LIN {X 0,Y 387.614,Z 136.056,A -85,B 0,C 180,E1 -14314.941,E2 -14314.941} C_VEL
LIN {X 0,Y 385.469,Z 134.733,A -85,B 0,C 180,E1 -14316.684,E2 -14316.684} C_VEL
LIN {X 0,Y 383.225,Z 132.712,A -85,B 0,C 180,E1 -14318.163,E2 -14318.163} C_VEL
LIN {X 0,Y 380.546,Z 129.667,A -85,B 0,C 180,E1 -14319.669,E2 -14319.669} C_VEL
LIN {X 0,Y 377.535,Z 127.903,A -85,B 0,C 180,E1 -14321.039,E2 -14321.039} C_VEL
LIN {X 0,Y 374.064,Z 124.674,A -85,B 0,C 180,E1 -14322.478,E2 -14322.478} C_VEL
LIN {X 0,Y 371.833,Z 122.319,A -85,B 0,C 180,E1 -14323.337,E2 -14323.337} C_VEL
LIN {X 0,Y 368.144,Z 119.325,A -85,B 0,C 180,E1 -14324.584,E2 -14324.584} C_VEL
LIN {X 0,Y 364.871,Z 115.734,A -85,B 0,C 180,E1 -14325.644,E2 -14325.644} C_VEL
LIN {X 0,Y 361.202,Z 112.484,A -85,B 0,C 180,E1 -14326.737,E2 -14326.737} C_VEL
LIN {X 0,Y 358.552,Z 109.441,A -85,B 0,C 180,E1 -14327.482,E2 -14327.482} C_VEL
LIN {X 0,Y 355.376,Z 106.45,A -85,B 0,C 180,E1 -14328.333,E2 -14328.333} C_VEL
LIN {X 0,Y 353.051,Z 103.518,A -85,B 0,C 180,E1 -14328.941,E2 -14328.941} C_VEL
LIN {X 0,Y 350.141,Z 100.557,A -85,B 0,C 180,E1 -14329.672,E2 -14329.672} C_VEL
LIN {X 0,Y 348.213,Z 97.966,A -85,B 0,C 180,E1 -14330.137,E2 -14330.137} C_VEL
LIN {X 0,Y 345.498,Z 95.057,A -85,B 0,C 180,E1 -14330.785,E2 -14330.785} C_VEL
LIN {X 0,Y 344.014,Z 92.683,A -85,B 0,C 180,E1 -14331.145,E2 -14331.145} C_VEL
LIN {X 0,Y 341.721,Z 90.357,A -85,B 0,C 180,E1 -14331.634,E2 -14331.634} C_VEL
LIN {X 0,Y 340.82,Z 88.079,A -85,B 0,C 180,E1 -14331.984,E2 -14331.984} C_VEL
LIN {X 0,Y 340.743,Z 87.555,A -85,B 0,C 180,E1 -14332.43,E2 -14332.43} C_VEL
LIN {X 0,Y 340.769,Z 87.54,A -85,B 0,C 180,E1 -14335.665,E2 -14335.665} C_VEL
LIN {X 0,Y 340.724,Z 87.528,A -85,B 0,C 180,E1 -14338.321,E2 -14338.321} C_VEL
LIN {X 0,Y 340.694,Z 87.545,A -85,B 0,C 180,E1 -14341.045,E2 -14341.045} C_VEL
LIN {X 0,Y 340.715,Z 87.514,A -85,B 0,C 180,E1 -14345.279,E2 -14345.279} C_VEL
LIN {X 0,Y 340.707,Z 87.545,A -85,B 0,C 180,E1 -14348.386,E2 -14348.386} C_VEL
LIN {X 0,Y 340.695,Z 87.5,A -85,B 0,C 180,E1 -14352.046,E2 -14352.046} C_VEL
LIN {X 0,Y 340.653,Z 87.551,A -85,B 0,C 180,E1 -14356.226,E2 -14356.226} C_VEL
LIN {X 0,Y 340.701,Z 87.535,A -85,B 0,C 180,E1 -14358.694,E2 -14358.694} C_VEL
LIN {X 0,Y 340.736,Z 87.543,A -85,B 0,C 180,E1 -14361.774,E2 -14361.774} C_VEL
LIN {X 0,Y 340.72,Z 87.526,A -85,B 0,C 180,E1 -14365.596,E2 -14365.596} C_VEL
LIN {X 0,Y 340.702,Z 87.543,A -85,B 0,C 180,E1 -14369.553,E2 -14369.553} C_VEL
LIN {X 0,Y 340.801,Z 87.511,A -85,B 0,C 180,E1 -14373.02,E2 -14373.02} C_VEL
LIN {X 0,Y 340.759,Z 87.528,A -85,B 0,C 180,E1 -14374.683,E2 -14374.683} C_VEL
LIN {X 0,Y 340.077,Z 87.623,A -85,B 0,C 180,E1 -14375.67,E2 -14375.67} C_VEL
LIN {X 0,Y 337.182,Z 87.982,A -85,B 0,C 180,E1 -14377.275,E2 -14377.275} C_VEL
LIN {X 0,Y 334.76,Z 88.277,A -85,B 0,C 180,E1 -14378.575,E2 -14378.575} C_VEL
LIN {X 0,Y 333.76,Z 88.394,A -85,B 0,C 180,E1 -14379.581,E2 -14379.581} C_VEL
LIN {X 0,Y 333.7,Z 88.393,A -85,B 0,C 180,E1 -14379.922,E2 -14379.922} C_VEL
LIN {X 0,Y 333.745,Z 88.397,A -85,B 0,C 180,E1 -14382.854,E2 -14382.854} C_VEL
LIN {X 0,Y 333.797,Z 88.402,A -85,B 0,C 180,E1 -14386.609,E2 -14386.609} C_VEL
LIN {X 0,Y 333.863,Z 88.365,A -85,B 0,C 180,E1 -14390.306,E2 -14390.306} C_VEL
LIN {X 0,Y 334.025,Z 88.368,A -85,B 0,C 180,E1 -14392.748,E2 -14392.748} C_VEL
LIN {X 0,Y 333.81,Z 88.402,A -85,B 0,C 180,E1 -14395.17,E2 -14395.17} C_VEL
LIN {X 0,Y 334.105,Z 88.355,A -85,B 0,C 180,E1 -14397.589,E2 -14397.589} C_VEL
LIN {X 0,Y 334.227,Z 88.319,A -85,B 0,C 180,E1 -14400.001,E2 -14400.001} C_VEL
LIN {X 0,Y 334.105,Z 88.356,A -85,B 0,C 180,E1 -14402.412,E2 -14402.412} C_VEL
LIN {X 0,Y 334.023,Z 88.374,A -85,B 0,C 180,E1 -14406.039,E2 -14406.039} C_VEL
LIN {X 0,Y 333.985,Z 88.358,A -85,B 0,C 180,E1 -14408.502,E2 -14408.502} C_VEL
LIN {X 0,Y 333.792,Z 88.395,A -85,B 0,C 180,E1 -14412.155,E2 -14412.155} C_VEL
LIN {X 0,Y 333.779,Z 88.399,A -85,B 0,C 180,E1 -14415.887,E2 -14415.887} C_VEL
LIN {X 0,Y 333.797,Z 88.374,A -85,B 0,C 180,E1 -14418.655,E2 -14418.655} C_VEL
LIN {X 0,Y 333.694,Z 88.414,A -85,B 0,C 180,E1 -14422.279,E2 -14422.279} C_VEL
LIN {X 0,Y 333.736,Z 88.392,A -85,B 0,C 180,E1 -14426.247,E2 -14426.247} C_VEL
LIN {X 0,Y 333.691,Z 88.409,A -85,B 0,C 180,E1 -14428.975,E2 -14428.975} C_VEL
LIN {X 0,Y 333.644,Z 88.417,A -85,B 0,C 180,E1 -14432.587,E2 -14432.587} C_VEL
LIN {X 0,Y 333.677,Z 88.415,A -85,B 0,C 180,E1 -14436.14,E2 -14436.14} C_VEL
LIN {X 0,Y 333.648,Z 88.414,A -85,B 0,C 180,E1 -14439.193,E2 -14439.193} C_VEL
LIN {X 0,Y 333.634,Z 88.428,A -85,B 0,C 180,E1 -14442.501,E2 -14442.501} C_VEL
LIN {X 0,Y 333.598,Z 88.427,A -85,B 0,C 180,E1 -14445.955,E2 -14445.955} C_VEL
LIN {X 0,Y 333.649,Z 88.399,A -85,B 0,C 180,E1 -14449.316,E2 -14449.316} C_VEL
LIN {X 0,Y 333.669,Z 88.419,A -85,B 0,C 180,E1 -14453.168,E2 -14453.168} C_VEL
LIN {X 0,Y 333.706,Z 88.483,A -85,B 0,C 180,E1 -14456.886,E2 -14456.886} C_VEL
LIN {X 0,Y 334.983,Z 94.79,A -85,B 0,C 180,E1 -14459.339,E2 -14459.339} C_VEL
LIN {X 0,Y 336.52,Z 102.522,A -85,B 0,C 180,E1 -14462.042,E2 -14462.042} C_VEL
LIN {X 0,Y 337.063,Z 107.291,A -85,B 0,C 180,E1 -14463.713,E2 -14463.713} C_VEL
LIN {X 0,Y 336.216,Z 114.217,A -85,B 0,C 180,E1 -14465.934,E2 -14465.934} C_VEL
LIN {X 0,Y 337.962,Z 122.359,A -85,B 0,C 180,E1 -14466.298,E2 -14466.298} C_VEL
LIN {X 0,Y 342.357,Z 144.864,A -85,B 0,C 180,E1 -14467.12,E2 -14467.12} C_VEL
LIN {X 0,Y 343.665,Z 153.202,A -85,B 0,C 180,E1 -14467.396,E2 -14467.396} C_VEL
LIN {X 0,Y 342.418,Z 218.942,A -85,B 0,C 180,E1 -14468.793,E2 -14468.793} C_VEL
LIN {X 0,Y 341.88,Z 229.679,A -85,B 0,C 180,E1 -14469.152,E2 -14469.152} C_VEL
LIN {X 0,Y 341.203,Z 238.778,A -85,B 0,C 180,E1 -14469.582,E2 -14469.582} C_VEL
LIN {X 0,Y 340.4,Z 248.132,A -85,B 0,C 180,E1 -14470.161,E2 -14470.161} C_VEL
LIN {X 0,Y 339.412,Z 258.273,A -85,B 0,C 180,E1 -14470.966,E2 -14470.966} C_VEL
LIN {X 0,Y 338.345,Z 267.266,A -85,B 0,C 180,E1 -14471.846,E2 -14471.846} C_VEL
LIN {X 0,Y 337.271,Z 275.994,A -85,B 0,C 180,E1 -14472.882,E2 -14472.882} C_VEL
LIN {X 0,Y 336.259,Z 283.752,A -85,B 0,C 180,E1 -14473.982,E2 -14473.982} C_VEL
LIN {X 0,Y 335.422,Z 290.636,A -85,B 0,C 180,E1 -14475.133,E2 -14475.133} C_VEL
LIN {X 0,Y 334.663,Z 296.812,A -85,B 0,C 180,E1 -14476.335,E2 -14476.335} C_VEL
LIN {X 0,Y 333.727,Z 303.347,A -85,B 0,C 180,E1 -14477.843,E2 -14477.843} C_VEL
LIN {X 0,Y 333.206,Z 307.85,A -85,B 0,C 180,E1 -14479.057,E2 -14479.057} C_VEL
LIN {X 0,Y 332.602,Z 313.342,A -85,B 0,C 180,E1 -14480.881,E2 -14480.881} C_VEL
LIN {X 0,Y 332.201,Z 317.667,A -85,B 0,C 180,E1 -14482.708,E2 -14482.708} C_VEL
LIN {X 0,Y 332.028,Z 320.418,A -85,B 0,C 180,E1 -14484.183,E2 -14484.183} C_VEL
LIN {X 0,Y 331.969,Z 323.224,A -85,B 0,C 180,E1 -14486.359,E2 -14486.359} C_VEL
LIN {X 0,Y 331.916,Z 324.281,A -85,B 0,C 180,E1 -14487.573,E2 -14487.573} C_VEL
LIN {X 0,Y 331.913,Z 324.87,A -85,B 0,C 180,E1 -14488.787,E2 -14488.787} C_VEL
LIN {X 0,Y 331.97,Z 325.026,A -85,B 0,C 180,E1 -14490,E2 -14490} C_VEL
LIN {X 0,Y 331.913,Z 324.87,A -85,B 0,C 180,E1 -14491.213,E2 -14491.213} C_VEL
LIN {X 0,Y 331.916,Z 324.281,A -85,B 0,C 180,E1 -14492.427,E2 -14492.427} C_VEL
LIN {X 0,Y 331.969,Z 321.835,A -85,B 0,C 180,E1 -14494.858,E2 -14494.858} C_VEL
LIN {X 0,Y 332.11,Z 318.884,A -85,B 0,C 180,E1 -14496.684,E2 -14496.684} C_VEL
LIN {X 0,Y 332.46,Z 314.897,A -85,B 0,C 180,E1 -14498.51,E2 -14498.51} C_VEL
LIN {X 0,Y 332.971,Z 309.766,A -85,B 0,C 180,E1 -14500.335,E2 -14500.335} C_VEL
LIN {X 0,Y 333.566,Z 304.502,A -85,B 0,C 180,E1 -14501.854,E2 -14501.854} C_VEL
LIN {X 0,Y 334.462,Z 298.188,A -85,B 0,C 180,E1 -14503.364,E2 -14503.364} C_VEL
LIN {X 0,Y 335.206,Z 292.235,A -85,B 0,C 180,E1 -14504.572,E2 -14504.572} C_VEL
LIN {X 0,Y 336.181,Z 285.31,A -85,B 0,C 180,E1 -14505.77,E2 -14505.77} C_VEL
LIN {X 0,Y 337.15,Z 277.129,A -85,B 0,C 180,E1 -14506.968,E2 -14506.968} C_VEL
LIN {X 0,Y 338.211,Z 268.619,A -85,B 0,C 180,E1 -14508.005,E2 -14508.005} C_VEL
LIN {X 0,Y 339.257,Z 259.905,A -85,B 0,C 180,E1 -14508.886,E2 -14508.886} C_VEL
LIN {X 0,Y 340.232,Z 250.147,A -85,B 0,C 180,E1 -14509.692,E2 -14509.692} C_VEL
LIN {X 0,Y 341.021,Z 241.354,A -85,B 0,C 180,E1 -14510.272,E2 -14510.272} C_VEL
LIN {X 0,Y 341.773,Z 231.427,A -85,B 0,C 180,E1 -14510.776,E2 -14510.776} C_VEL
LIN {X 0,Y 342.274,Z 221.571,A -85,B 0,C 180,E1 -14511.138,E2 -14511.138} C_VEL
LIN {X 0,Y 342.869,Z 198.751,A -85,B 0,C 180,E1 -14511.651,E2 -14511.651} C_VEL
LIN {X 0,Y 343.58,Z 152.553,A -85,B 0,C 180,E1 -14512.624,E2 -14512.624} C_VEL
LIN {X 0,Y 339.442,Z 129.203,A -85,B 0,C 180,E1 -14513.439,E2 -14513.439} C_VEL
LIN {X 0,Y 336.241,Z 114.522,A -85,B 0,C 180,E1 -14514.032,E2 -14514.032} C_VEL
LIN {X 0,Y 336.325,Z 112.923,A -85,B 0,C 180,E1 -14514.408,E2 -14514.408} C_VEL
LIN {X 0,Y 337.068,Z 107.285,A -85,B 0,C 180,E1 -14516.288,E2 -14516.288} C_VEL
LIN {X 0,Y 336.514,Z 102.53,A -85,B 0,C 180,E1 -14517.956,E2 -14517.956} C_VEL
LIN {X 0,Y 334.834,Z 93.824,A -85,B 0,C 180,E1 -14521.091,E2 -14521.091} C_VEL
LIN {X 0,Y 333.676,Z 88.433,A -85,B 0,C 180,E1 -14523.161,E2 -14523.161} C_VEL
LIN {X 0,Y 333.669,Z 88.419,A -85,B 0,C 180,E1 -14526.832,E2 -14526.832} C_VEL
LIN {X 0,Y 333.648,Z 88.4,A -85,B 0,C 180,E1 -14530.767,E2 -14530.767} C_VEL
LIN {X 0,Y 333.595,Z 88.428,A -85,B 0,C 180,E1 -14534.25,E2 -14534.25} C_VEL
LIN {X 0,Y 333.643,Z 88.426,A -85,B 0,C 180,E1 -14537.618,E2 -14537.618} C_VEL
LIN {X 0,Y 333.654,Z 88.417,A -85,B 0,C 180,E1 -14541.202,E2 -14541.202} C_VEL
LIN {X 0,Y 333.677,Z 88.415,A -85,B 0,C 180,E1 -14543.86,E2 -14543.86} C_VEL
LIN {X 0,Y 333.644,Z 88.417,A -85,B 0,C 180,E1 -14547.413,E2 -14547.413} C_VEL
LIN {X 0,Y 333.691,Z 88.409,A -85,B 0,C 180,E1 -14551.025,E2 -14551.025} C_VEL
LIN {X 0,Y 333.736,Z 88.392,A -85,B 0,C 180,E1 -14553.753,E2 -14553.753} C_VEL
LIN {X 0,Y 333.721,Z 88.411,A -85,B 0,C 180,E1 -14557.913,E2 -14557.913} C_VEL
LIN {X 0,Y 333.794,Z 88.375,A -85,B 0,C 180,E1 -14561.589,E2 -14561.589} C_VEL
LIN {X 0,Y 333.809,Z 88.4,A -85,B 0,C 180,E1 -14565.576,E2 -14565.576} C_VEL
LIN {X 0,Y 333.834,Z 88.376,A -85,B 0,C 180,E1 -14569.077,E2 -14569.077} C_VEL
LIN {X 0,Y 334.027,Z 88.366,A -85,B 0,C 180,E1 -14572.747,E2 -14572.747} C_VEL
LIN {X 0,Y 333.812,Z 88.402,A -85,B 0,C 180,E1 -14575.168,E2 -14575.168} C_VEL
LIN {X 0,Y 334.105,Z 88.356,A -85,B 0,C 180,E1 -14577.588,E2 -14577.588} C_VEL
LIN {X 0,Y 334.227,Z 88.319,A -85,B 0,C 180,E1 -14579.999,E2 -14579.999} C_VEL
LIN {X 0,Y 334.105,Z 88.355,A -85,B 0,C 180,E1 -14582.411,E2 -14582.411} C_VEL
LIN {X 0,Y 334.025,Z 88.368,A -85,B 0,C 180,E1 -14587.252,E2 -14587.252} C_VEL
LIN {X 0,Y 333.836,Z 88.376,A -85,B 0,C 180,E1 -14590.921,E2 -14590.921} C_VEL
LIN {X 0,Y 333.807,Z 88.403,A -85,B 0,C 180,E1 -14594.634,E2 -14594.634} C_VEL
LIN {X 0,Y 333.794,Z 88.378,A -85,B 0,C 180,E1 -14598.654,E2 -14598.654} C_VEL
LIN {X 0,Y 333.691,Z 88.416,A -85,B 0,C 180,E1 -14602.278,E2 -14602.278} C_VEL
LIN {X 0,Y 333.733,Z 88.397,A -85,B 0,C 180,E1 -14606.246,E2 -14606.246} C_VEL
LIN {X 0,Y 333.687,Z 88.408,A -85,B 0,C 180,E1 -14608.973,E2 -14608.973} C_VEL
LIN {X 0,Y 333.64,Z 88.42,A -85,B 0,C 180,E1 -14612.586,E2 -14612.586} C_VEL
LIN {X 0,Y 333.674,Z 88.414,A -85,B 0,C 180,E1 -14616.138,E2 -14616.138} C_VEL
LIN {X 0,Y 333.669,Z 88.415,A -85,B 0,C 180,E1 -14619.188,E2 -14619.188} C_VEL
LIN {X 0,Y 333.657,Z 88.421,A -85,B 0,C 180,E1 -14622.505,E2 -14622.505} C_VEL
LIN {X 0,Y 333.593,Z 88.405,A -85,B 0,C 180,E1 -14625.955,E2 -14625.955} C_VEL
LIN {X 0,Y 333.643,Z 88.39,A -85,B 0,C 180,E1 -14629.315,E2 -14629.315} C_VEL
LIN {X 0,Y 333.662,Z 88.419,A -85,B 0,C 180,E1 -14633.167,E2 -14633.167} C_VEL
LIN {X 0,Y 333.67,Z 88.39,A -85,B 0,C 180,E1 -14635.341,E2 -14635.341} C_VEL
LIN {X 0,Y 333.686,Z 88.405,A -85,B 0,C 180,E1 -14639.637,E2 -14639.637} C_VEL
LIN {X 0,Y 333.736,Z 88.41,A -85,B 0,C 180,E1 -14642.401,E2 -14642.401} C_VEL
LIN {X 0,Y 333.723,Z 88.417,A -85,B 0,C 180,E1 -14645.091,E2 -14645.091} C_VEL
LIN {X 0,Y 333.715,Z 88.563,A -85,B 0,C 180,E1 -14646.635,E2 -14646.635} C_VEL
LIN {X 0,Y 333.903,Z 89.473,A -85,B 0,C 180,E1 -14646.906,E2 -14646.906} C_VEL
LIN {X 0,Y 335.441,Z 92.245,A -85,B 0,C 180,E1 -14647.293,E2 -14647.293} C_VEL
LIN {X 0,Y 337.24,Z 94.134,A -85,B 0,C 180,E1 -14647.649,E2 -14647.649} C_VEL
LIN {X 0,Y 339.457,Z 97.377,A -85,B 0,C 180,E1 -14648.16,E2 -14648.16} C_VEL
LIN {X 0,Y 341.244,Z 99.3,A -85,B 0,C 180,E1 -14648.55,E2 -14648.55} C_VEL
LIN {X 0,Y 344.183,Z 103.016,A -85,B 0,C 180,E1 -14649.205,E2 -14649.205} C_VEL
LIN {X 0,Y 346.131,Z 105.087,A -85,B 0,C 180,E1 -14649.669,E2 -14649.669} C_VEL
LIN {X 0,Y 349.254,Z 108.734,A -85,B 0,C 180,E1 -14650.409,E2 -14650.409} C_VEL
LIN {X 0,Y 351.181,Z 110.612,A -85,B 0,C 180,E1 -14650.88,E2 -14650.88} C_VEL
LIN {X 0,Y 354.741,Z 114.632,A -85,B 0,C 180,E1 -14651.8,E2 -14651.8} C_VEL
LIN {X 0,Y 357.121,Z 116.838,A -85,B 0,C 180,E1 -14652.431,E2 -14652.431} C_VEL
LIN {X 0,Y 361.089,Z 120.94,A -85,B 0,C 180,E1 -14653.544,E2 -14653.544} C_VEL
LIN {X 0,Y 363.83,Z 123.291,A -85,B 0,C 180,E1 -14654.364,E2 -14654.364} C_VEL
LIN {X 0,Y 367.524,Z 127.112,A -85,B 0,C 180,E1 -14655.553,E2 -14655.553} C_VEL
LIN {X 0,Y 371.229,Z 130.062,A -85,B 0,C 180,E1 -14656.813,E2 -14656.813} C_VEL
LIN {X 0,Y 374.888,Z 133.747,A -85,B 0,C 180,E1 -14658.241,E2 -14658.241} C_VEL
LIN {X 0,Y 378.478,Z 136.219,A -85,B 0,C 180,E1 -14659.786,E2 -14659.786} C_VEL
LIN {X 0,Y 379.78,Z 137.046,A -85,B 0,C 180,E1 -14660.413,E2 -14660.413} C_VEL
LIN {X 0,Y 382.384,Z 139.979,A -85,B 0,C 180,E1 -14661.881,E2 -14661.881} C_VEL
LIN {X 0,Y 384.713,Z 141.903,A -85,B 0,C 180,E1 -14663.407,E2 -14663.407} C_VEL
LIN {X 0,Y 387.037,Z 143.23,A -85,B 0,C 180,E1 -14665.318,E2 -14665.318} C_VEL
LIN {X 0,Y 388.665,Z 143.823,A -85,B 0,C 180,E1 -14667.428,E2 -14667.428} C_VEL
LIN {X 0,Y 389.264,Z 144.277,A -85,B 0,C 180,E1 -14668.965,E2 -14668.965} C_VEL
LIN {X 0,Y 389.407,Z 144.179,A -85,B 0,C 180,E1 -14670,E2 -14670} C_VEL
LIN {X 0,Y 389.126,Z 144.135,A -85,B 0,C 180,E1 -14671.552,E2 -14671.552} C_VEL
LIN {X 0,Y 388.36,Z 143.701,A -85,B 0,C 180,E1 -14673.112,E2 -14673.112} C_VEL
LIN {X 0,Y 386.736,Z 143.092,A -85,B 0,C 180,E1 -14674.943,E2 -14674.943} C_VEL
LIN {X 0,Y 384.56,Z 141.783,A -85,B 0,C 180,E1 -14676.7,E2 -14676.7} C_VEL
LIN {X 0,Y 382.221,Z 139.834,A -85,B 0,C 180,E1 -14678.214,E2 -14678.214} C_VEL
LIN {X 0,Y 379.214,Z 136.56,A -85,B 0,C 180,E1 -14679.864,E2 -14679.864} C_VEL
LIN {X 0,Y 376.134,Z 134.752,A -85,B 0,C 180,E1 -14681.228,E2 -14681.228} C_VEL
LIN {X 0,Y 372.666,Z 131.662,A -85,B 0,C 180,E1 -14682.629,E2 -14682.629} C_VEL
LIN {X 0,Y 370.003,Z 128.94,A -85,B 0,C 180,E1 -14683.635,E2 -14683.635} C_VEL
LIN {X 0,Y 366.039,Z 125.687,A -85,B 0,C 180,E1 -14684.945,E2 -14684.945} C_VEL
LIN {X 0,Y 362.682,Z 122.188,A -85,B 0,C 180,E1 -14685.986,E2 -14685.986} C_VEL
LIN {X 0,Y 358.732,Z 118.722,A -85,B 0,C 180,E1 -14687.109,E2 -14687.109} C_VEL
LIN {X 0,Y 355.813,Z 115.508,A -85,B 0,C 180,E1 -14687.929,E2 -14687.929} C_VEL
LIN {X 0,Y 352.189,Z 111.983,A -85,B 0,C 180,E1 -14688.848,E2 -14688.848} C_VEL
LIN {X 0,Y 350.013,Z 109.386,A -85,B 0,C 180,E1 -14689.415,E2 -14689.415} C_VEL
LIN {X 0,Y 346.456,Z 105.581,A -85,B 0,C 180,E1 -14690.25,E2 -14690.25} C_VEL
LIN {X 0,Y 344.965,Z 103.745,A -85,B 0,C 180,E1 -14690.614,E2 -14690.614} C_VEL
LIN {X 0,Y 341.952,Z 100.422,A -85,B 0,C 180,E1 -14691.286,E2 -14691.286} C_VEL
LIN {X 0,Y 340.285,Z 98.185,A -85,B 0,C 180,E1 -14691.661,E2 -14691.661} C_VEL
LIN {X 0,Y 337.761,Z 95.054,A -85,B 0,C 180,E1 -14692.231,E2 -14692.231} C_VEL
LIN {X 0,Y 336.543,Z 93.281,A -85,B 0,C 180,E1 -14692.493,E2 -14692.493} C_VEL
LIN {X 0,Y 334.617,Z 91.122,A -85,B 0,C 180,E1 -14692.878,E2 -14692.878} C_VEL
LIN {X 0,Y 333.802,Z 89.069,A -85,B 0,C 180,E1 -14693.171,E2 -14693.171} C_VEL
LIN {X 0,Y 333.68,Z 88.493,A -85,B 0,C 180,E1 -14693.425,E2 -14693.425} C_VEL
LIN {X 0,Y 333.731,Z 88.416,A -85,B 0,C 180,E1 -14696.247,E2 -14696.247} C_VEL
LIN {X 0,Y 333.686,Z 88.399,A -85,B 0,C 180,E1 -14698.974,E2 -14698.974} C_VEL
LIN {X 0,Y 333.64,Z 88.421,A -85,B 0,C 180,E1 -14702.587,E2 -14702.587} C_VEL
LIN {X 0,Y 333.673,Z 88.401,A -85,B 0,C 180,E1 -14706.139,E2 -14706.139} C_VEL
LIN {X 0,Y 333.643,Z 88.418,A -85,B 0,C 180,E1 -14709.193,E2 -14709.193} C_VEL
LIN {X 0,Y 333.628,Z 88.381,A -85,B 0,C 180,E1 -14712.5,E2 -14712.5} C_VEL
LIN {X 0,Y 333.597,Z 88.431,A -85,B 0,C 180,E1 -14715.956,E2 -14715.956} C_VEL
LIN {X 0,Y 333.653,Z 88.41,A -85,B 0,C 180,E1 -14719.314,E2 -14719.314} C_VEL
LIN {X 0,Y 333.653,Z 88.424,A -85,B 0,C 180,E1 -14722.35,E2 -14722.35} C_VEL
LIN {X 0,Y 333.671,Z 88.403,A -85,B 0,C 180,E1 -14725.342,E2 -14725.342} C_VEL
LIN {X 0,Y 333.688,Z 88.418,A -85,B 0,C 180,E1 -14729.638,E2 -14729.638} C_VEL
LIN {X 0,Y 333.737,Z 88.391,A -85,B 0,C 180,E1 -14732.401,E2 -14732.401} C_VEL
LIN {X 0,Y 333.725,Z 88.409,A -85,B 0,C 180,E1 -14735.091,E2 -14735.091} C_VEL
LIN {X 0,Y 333.678,Z 88.407,A -85,B 0,C 180,E1 -14739.02,E2 -14739.02} C_VEL
LIN {X 0,Y 333.7,Z 88.393,A -85,B 0,C 180,E1 -14739.922,E2 -14739.922} C_VEL
LIN {X 0,Y 333.09,Z 88.468,A -85,B 0,C 180,E1 -14740.929,E2 -14740.929} C_VEL
LIN {X 0,Y 330.266,Z 88.832,A -85,B 0,C 180,E1 -14742.568,E2 -14742.568} C_VEL
LIN {X 0,Y 327.852,Z 89.143,A -85,B 0,C 180,E1 -14743.896,E2 -14743.896} C_VEL
LIN {X 0,Y 326.83,Z 89.274,A -85,B 0,C 180,E1 -14744.924,E2 -14744.924} C_VEL
LIN {X 0,Y 326.756,Z 89.282,A -85,B 0,C 180,E1 -14745.272,E2 -14745.272} C_VEL
LIN {X 0,Y 326.772,Z 89.256,A -85,B 0,C 180,E1 -14748.84,E2 -14748.84} C_VEL
LIN {X 0,Y 326.979,Z 89.242,A -85,B 0,C 180,E1 -14752.591,E2 -14752.591} C_VEL
LIN {X 0,Y 326.777,Z 89.278,A -85,B 0,C 180,E1 -14755.066,E2 -14755.066} C_VEL
LIN {X 0,Y 327.046,Z 89.234,A -85,B 0,C 180,E1 -14757.537,E2 -14757.537} C_VEL
LIN {X 0,Y 327.179,Z 89.196,A -85,B 0,C 180,E1 -14760.001,E2 -14760.001} C_VEL
LIN {X 0,Y 327.046,Z 89.236,A -85,B 0,C 180,E1 -14762.464,E2 -14762.464} C_VEL
LIN {X 0,Y 326.999,Z 89.247,A -85,B 0,C 180,E1 -14766.17,E2 -14766.17} C_VEL
LIN {X 0,Y 326.915,Z 89.236,A -85,B 0,C 180,E1 -14768.656,E2 -14768.656} C_VEL
LIN {X 0,Y 326.736,Z 89.277,A -85,B 0,C 180,E1 -14772.422,E2 -14772.422} C_VEL
LIN {X 0,Y 326.755,Z 89.28,A -85,B 0,C 180,E1 -14774.958,E2 -14774.958} C_VEL
LIN {X 0,Y 326.733,Z 89.253,A -85,B 0,C 180,E1 -14778.839,E2 -14778.839} C_VEL
LIN {X 0,Y 326.622,Z 89.297,A -85,B 0,C 180,E1 -14782.788,E2 -14782.788} C_VEL
LIN {X 0,Y 326.691,Z 89.274,A -85,B 0,C 180,E1 -14785.484,E2 -14785.484} C_VEL
LIN {X 0,Y 326.649,Z 89.295,A -85,B 0,C 180,E1 -14789.661,E2 -14789.661} C_VEL
LIN {X 0,Y 326.608,Z 89.28,A -85,B 0,C 180,E1 -14794.02,E2 -14794.02} C_VEL
LIN {X 0,Y 326.629,Z 89.299,A -85,B 0,C 180,E1 -14797.239,E2 -14797.239} C_VEL
LIN {X 0,Y 326.579,Z 89.297,A -85,B 0,C 180,E1 -14801.132,E2 -14801.132} C_VEL
LIN {X 0,Y 326.529,Z 89.303,A -85,B 0,C 180,E1 -14804.743,E2 -14804.743} C_VEL
LIN {X 0,Y 326.578,Z 89.293,A -85,B 0,C 180,E1 -14808.155,E2 -14808.155} C_VEL
LIN {X 0,Y 326.627,Z 89.285,A -85,B 0,C 180,E1 -14811.392,E2 -14811.392} C_VEL
LIN {X 0,Y 326.622,Z 89.283,A -85,B 0,C 180,E1 -14814.852,E2 -14814.852} C_VEL
LIN {X 0,Y 326.676,Z 89.534,A -85,B 0,C 180,E1 -14816.565,E2 -14816.565} C_VEL
LIN {X 0,Y 328.195,Z 96.942,A -85,B 0,C 180,E1 -14819.431,E2 -14819.431} C_VEL
LIN {X 0,Y 329.614,Z 104.093,A -85,B 0,C 180,E1 -14822.025,E2 -14822.025} C_VEL
LIN {X 0,Y 330.081,Z 108.039,A -85,B 0,C 180,E1 -14823.441,E2 -14823.441} C_VEL
LIN {X 0,Y 329.381,Z 113.892,A -85,B 0,C 180,E1 -14825.38,E2 -14825.38} C_VEL
LIN {X 0,Y 330.25,Z 118.246,A -85,B 0,C 180,E1 -14825.619,E2 -14825.619} C_VEL
LIN {X 0,Y 334.159,Z 136.803,A -85,B 0,C 180,E1 -14826.346,E2 -14826.346} C_VEL
LIN {X 0,Y 337.096,Z 153.67,A -85,B 0,C 180,E1 -14826.945,E2 -14826.945} C_VEL
LIN {X 0,Y 335.823,Z 218.758,A -85,B 0,C 180,E1 -14828.355,E2 -14828.355} C_VEL
LIN {X 0,Y 335.27,Z 229.489,A -85,B 0,C 180,E1 -14828.721,E2 -14828.721} C_VEL
LIN {X 0,Y 334.563,Z 238.588,A -85,B 0,C 180,E1 -14829.158,E2 -14829.158} C_VEL
LIN {X 0,Y 333.747,Z 247.942,A -85,B 0,C 180,E1 -14829.749,E2 -14829.749} C_VEL
LIN {X 0,Y 332.703,Z 258.082,A -85,B 0,C 180,E1 -14830.567,E2 -14830.567} C_VEL
LIN {X 0,Y 331.594,Z 267.076,A -85,B 0,C 180,E1 -14831.463,E2 -14831.463} C_VEL
LIN {X 0,Y 330.473,Z 275.803,A -85,B 0,C 180,E1 -14832.519,E2 -14832.519} C_VEL
LIN {X 0,Y 329.484,Z 283.197,A -85,B 0,C 180,E1 -14833.583,E2 -14833.583} C_VEL
LIN {X 0,Y 328.52,Z 290.62,A -85,B 0,C 180,E1 -14834.847,E2 -14834.847} C_VEL
LIN {X 0,Y 327.75,Z 296.621,A -85,B 0,C 180,E1 -14836.041,E2 -14836.041} C_VEL
LIN {X 0,Y 326.766,Z 303.156,A -85,B 0,C 180,E1 -14837.58,E2 -14837.58} C_VEL
LIN {X 0,Y 326.18,Z 307.658,A -85,B 0,C 180,E1 -14838.819,E2 -14838.819} C_VEL
LIN {X 0,Y 325.57,Z 313.151,A -85,B 0,C 180,E1 -14840.683,E2 -14840.683} C_VEL
LIN {X 0,Y 325.153,Z 317.477,A -85,B 0,C 180,E1 -14842.549,E2 -14842.549} C_VEL
LIN {X 0,Y 324.92,Z 320.521,A -85,B 0,C 180,E1 -14844.259,E2 -14844.259} C_VEL
LIN {X 0,Y 324.876,Z 323.033,A -85,B 0,C 180,E1 -14846.279,E2 -14846.279} C_VEL
LIN {X 0,Y 324.835,Z 324.091,A -85,B 0,C 180,E1 -14847.52,E2 -14847.52} C_VEL
LIN {X 0,Y 324.822,Z 324.68,A -85,B 0,C 180,E1 -14848.76,E2 -14848.76} C_VEL
LIN {X 0,Y 324.874,Z 324.836,A -85,B 0,C 180,E1 -14850,E2 -14850} C_VEL
LIN {X 0,Y 324.822,Z 324.68,A -85,B 0,C 180,E1 -14851.24,E2 -14851.24} C_VEL
LIN {X 0,Y 324.835,Z 324.091,A -85,B 0,C 180,E1 -14852.48,E2 -14852.48} C_VEL
LIN {X 0,Y 324.88,Z 321.644,A -85,B 0,C 180,E1 -14854.964,E2 -14854.964} C_VEL
LIN {X 0,Y 325.049,Z 318.694,A -85,B 0,C 180,E1 -14856.83,E2 -14856.83} C_VEL
LIN {X 0,Y 325.4,Z 314.705,A -85,B 0,C 180,E1 -14858.696,E2 -14858.696} C_VEL
LIN {X 0,Y 325.948,Z 309.574,A -85,B 0,C 180,E1 -14860.561,E2 -14860.561} C_VEL
LIN {X 0,Y 326.601,Z 304.311,A -85,B 0,C 180,E1 -14862.111,E2 -14862.111} C_VEL
LIN {X 0,Y 327.541,Z 297.997,A -85,B 0,C 180,E1 -14863.652,E2 -14863.652} C_VEL
LIN {X 0,Y 328.313,Z 292.044,A -85,B 0,C 180,E1 -14864.885,E2 -14864.885} C_VEL
LIN {X 0,Y 329.28,Z 285.118,A -85,B 0,C 180,E1 -14866.109,E2 -14866.109} C_VEL
LIN {X 0,Y 330.323,Z 276.937,A -85,B 0,C 180,E1 -14867.329,E2 -14867.329} C_VEL
LIN {X 0,Y 331.444,Z 268.428,A -85,B 0,C 180,E1 -14868.386,E2 -14868.386} C_VEL
LIN {X 0,Y 332.545,Z 259.714,A -85,B 0,C 180,E1 -14869.282,E2 -14869.282} C_VEL
LIN {X 0,Y 333.565,Z 249.957,A -85,B 0,C 180,E1 -14870.102,E2 -14870.102} C_VEL
LIN {X 0,Y 334.388,Z 241.164,A -85,B 0,C 180,E1 -14870.693,E2 -14870.693} C_VEL
LIN {X 0,Y 335.151,Z 231.237,A -85,B 0,C 180,E1 -14871.206,E2 -14871.206} C_VEL
LIN {X 0,Y 335.667,Z 221.381,A -85,B 0,C 180,E1 -14871.575,E2 -14871.575} C_VEL
LIN {X 0,Y 336.282,Z 198.56,A -85,B 0,C 180,E1 -14872.097,E2 -14872.097} C_VEL
LIN {X 0,Y 337.047,Z 153.551,A -85,B 0,C 180,E1 -14873.061,E2 -14873.061} C_VEL
LIN {X 0,Y 333.076,Z 131.136,A -85,B 0,C 180,E1 -14873.865,E2 -14873.865} C_VEL
LIN {X 0,Y 329.428,Z 114.114,A -85,B 0,C 180,E1 -14874.583,E2 -14874.583} C_VEL
LIN {X 0,Y 329.614,Z 111.881,A -85,B 0,C 180,E1 -14875.242,E2 -14875.242} C_VEL
LIN {X 0,Y 330.099,Z 107.941,A -85,B 0,C 180,E1 -14876.592,E2 -14876.592} C_VEL
LIN {X 0,Y 329.139,Z 101.587,A -85,B 0,C 180,E1 -14878.899,E2 -14878.899} C_VEL
LIN {X 0,Y 327.224,Z 92.007,A -85,B 0,C 180,E1 -14882.475,E2 -14882.475} C_VEL
LIN {X 0,Y 326.631,Z 89.312,A -85,B 0,C 180,E1 -14883.584,E2 -14883.584} C_VEL
LIN {X 0,Y 326.632,Z 89.299,A -85,B 0,C 180,E1 -14887.239,E2 -14887.239} C_VEL
LIN {X 0,Y 326.579,Z 89.283,A -85,B 0,C 180,E1 -14891.131,E2 -14891.131} C_VEL
LIN {X 0,Y 326.529,Z 89.305,A -85,B 0,C 180,E1 -14894.742,E2 -14894.742} C_VEL
LIN {X 0,Y 326.578,Z 89.303,A -85,B 0,C 180,E1 -14898.154,E2 -14898.154} C_VEL
LIN {X 0,Y 326.625,Z 89.295,A -85,B 0,C 180,E1 -14901.391,E2 -14901.391} C_VEL
LIN {X 0,Y 326.621,Z 89.284,A -85,B 0,C 180,E1 -14904.851,E2 -14904.851} C_VEL
LIN {X 0,Y 326.609,Z 89.294,A -85,B 0,C 180,E1 -14907.455,E2 -14907.455} C_VEL
LIN {X 0,Y 326.649,Z 89.295,A -85,B 0,C 180,E1 -14910.339,E2 -14910.339} C_VEL
LIN {X 0,Y 326.691,Z 89.274,A -85,B 0,C 180,E1 -14914.516,E2 -14914.516} C_VEL
LIN {X 0,Y 326.647,Z 89.288,A -85,B 0,C 180,E1 -14918.545,E2 -14918.545} C_VEL
LIN {X 0,Y 326.745,Z 89.251,A -85,B 0,C 180,E1 -14921.177,E2 -14921.177} C_VEL
LIN {X 0,Y 326.764,Z 89.278,A -85,B 0,C 180,E1 -14925.432,E2 -14925.432} C_VEL
LIN {X 0,Y 326.77,Z 89.257,A -85,B 0,C 180,E1 -14928.838,E2 -14928.838} C_VEL
LIN {X 0,Y 326.981,Z 89.24,A -85,B 0,C 180,E1 -14932.59,E2 -14932.59} C_VEL
LIN {X 0,Y 326.779,Z 89.278,A -85,B 0,C 180,E1 -14935.064,E2 -14935.064} C_VEL
LIN {X 0,Y 327.046,Z 89.236,A -85,B 0,C 180,E1 -14937.536,E2 -14937.536} C_VEL
LIN {X 0,Y 327.179,Z 89.196,A -85,B 0,C 180,E1 -14939.999,E2 -14939.999} C_VEL
LIN {X 0,Y 327.046,Z 89.234,A -85,B 0,C 180,E1 -14942.463,E2 -14942.463} C_VEL
LIN {X 0,Y 326.971,Z 89.246,A -85,B 0,C 180,E1 -14946.654,E2 -14946.654} C_VEL
LIN {X 0,Y 326.814,Z 89.242,A -85,B 0,C 180,E1 -14949.906,E2 -14949.906} C_VEL
LIN {X 0,Y 326.759,Z 89.283,A -85,B 0,C 180,E1 -14953.685,E2 -14953.685} C_VEL
LIN {X 0,Y 326.697,Z 89.27,A -85,B 0,C 180,E1 -14957.527,E2 -14957.527} C_VEL
LIN {X 0,Y 326.661,Z 89.273,A -85,B 0,C 180,E1 -14960.134,E2 -14960.134} C_VEL
LIN {X 0,Y 326.65,Z 89.293,A -85,B 0,C 180,E1 -14964.128,E2 -14964.128} C_VEL
LIN {X 0,Y 326.68,Z 89.269,A -85,B 0,C 180,E1 -14966.857,E2 -14966.857} C_VEL
LIN {X 0,Y 326.631,Z 89.298,A -85,B 0,C 180,E1 -14970.609,E2 -14970.609} C_VEL
LIN {X 0,Y 326.604,Z 89.284,A -85,B 0,C 180,E1 -14974.019,E2 -14974.019} C_VEL
LIN {X 0,Y 326.627,Z 89.301,A -85,B 0,C 180,E1 -14977.239,E2 -14977.239} C_VEL
LIN {X 0,Y 326.601,Z 89.289,A -85,B 0,C 180,E1 -14980.207,E2 -14980.207} C_VEL
LIN {X 0,Y 326.569,Z 89.305,A -85,B 0,C 180,E1 -14983.523,E2 -14983.523} C_VEL
LIN {X 0,Y 326.572,Z 89.262,A -85,B 0,C 180,E1 -14987.028,E2 -14987.028} C_VEL
LIN {X 0,Y 326.608,Z 89.293,A -85,B 0,C 180,E1 -14990.772,E2 -14990.772} C_VEL
LIN {X 0,Y 326.609,Z 89.274,A -85,B 0,C 180,E1 -14994.48,E2 -14994.48} C_VEL
LIN {X 0,Y 326.604,Z 89.297,A -85,B 0,C 180,E1 -14997.455,E2 -14997.455} C_VEL
LIN {X 0,Y 326.644,Z 89.276,A -85,B 0,C 180,E1 -15000.339,E2 -15000.339} C_VEL
LIN {X 0,Y 326.686,Z 89.293,A -85,B 0,C 180,E1 -15004.516,E2 -15004.516} C_VEL
LIN {X 0,Y 326.692,Z 89.586,A -85,B 0,C 180,E1 -15005.621,E2 -15005.621} C_VEL
LIN {X 0,Y 326.998,Z 90.818,A -85,B 0,C 180,E1 -15005.854,E2 -15005.854} C_VEL
LIN {X 0,Y 328.543,Z 93.352,A -85,B 0,C 180,E1 -15006.172,E2 -15006.172} C_VEL
LIN {X 0,Y 329.922,Z 94.854,A -85,B 0,C 180,E1 -15006.429,E2 -15006.429} C_VEL
LIN {X 0,Y 332.332,Z 98.356,A -85,B 0,C 180,E1 -15006.946,E2 -15006.946} C_VEL
LIN {X 0,Y 333.985,Z 100.385,A -85,B 0,C 180,E1 -15007.286,E2 -15007.286} C_VEL
LIN {X 0,Y 336.999,Z 103.96,A -85,B 0,C 180,E1 -15007.902,E2 -15007.902} C_VEL
LIN {X 0,Y 341.329,Z 109.194,A -85,B 0,C 180,E1 -15008.866,E2 -15008.866} C_VEL
LIN {X 0,Y 343.414,Z 111.467,A -85,B 0,C 180,E1 -15009.321,E2 -15009.321} C_VEL
LIN {X 0,Y 347.347,Z 115.644,A -85,B 0,C 180,E1 -15010.249,E2 -15010.249} C_VEL
LIN {X 0,Y 352.042,Z 120.78,A -85,B 0,C 180,E1 -15011.415,E2 -15011.415} C_VEL
LIN {X 0,Y 354.866,Z 123.383,A -85,B 0,C 180,E1 -15012.126,E2 -15012.126} C_VEL
LIN {X 0,Y 359.165,Z 127.608,A -85,B 0,C 180,E1 -15013.306,E2 -15013.306} C_VEL
LIN {X 0,Y 361.767,Z 129.841,A -85,B 0,C 180,E1 -15014.059,E2 -15014.059} C_VEL
LIN {X 0,Y 365.634,Z 133.693,A -85,B 0,C 180,E1 -15015.257,E2 -15015.257} C_VEL
LIN {X 0,Y 369.613,Z 136.87,A -85,B 0,C 180,E1 -15016.584,E2 -15016.584} C_VEL
LIN {X 0,Y 373.52,Z 140.631,A -85,B 0,C 180,E1 -15018.07,E2 -15018.07} C_VEL
LIN {X 0,Y 377.406,Z 143.221,A -85,B 0,C 180,E1 -15019.711,E2 -15019.711} C_VEL
LIN {X 0,Y 378.643,Z 144.141,A -85,B 0,C 180,E1 -15020.316,E2 -15020.316} C_VEL
LIN {X 0,Y 381.247,Z 146.957,A -85,B 0,C 180,E1 -15021.75,E2 -15021.75} C_VEL
LIN {X 0,Y 383.646,Z 148.872,A -85,B 0,C 180,E1 -15023.284,E2 -15023.284} C_VEL
LIN {X 0,Y 385.845,Z 150.137,A -85,B 0,C 180,E1 -15025.046,E2 -15025.046} C_VEL
LIN {X 0,Y 387.489,Z 150.712,A -85,B 0,C 180,E1 -15026.881,E2 -15026.881} C_VEL
LIN {X 0,Y 388.398,Z 151.323,A -85,B 0,C 180,E1 -15028.963,E2 -15028.963} C_VEL
LIN {X 0,Y 388.542,Z 151.227,A -85,B 0,C 180,E1 -15030,E2 -15030} C_VEL
LIN {X 0,Y 388.258,Z 151.183,A -85,B 0,C 180,E1 -15031.556,E2 -15031.556} C_VEL
LIN {X 0,Y 387.234,Z 150.668,A -85,B 0,C 180,E1 -15033.443,E2 -15033.443} C_VEL
LIN {X 0,Y 385.526,Z 149.996,A -85,B 0,C 180,E1 -15035.23,E2 -15035.23} C_VEL
LIN {X 0,Y 383.275,Z 148.615,A -85,B 0,C 180,E1 -15036.978,E2 -15036.978} C_VEL
LIN {X 0,Y 380.457,Z 146.181,A -85,B 0,C 180,E1 -15038.725,E2 -15038.725} C_VEL
LIN {X 0,Y 377.888,Z 143.449,A -85,B 0,C 180,E1 -15040.06,E2 -15040.06} C_VEL
LIN {X 0,Y 374.225,Z 141.197,A -85,B 0,C 180,E1 -15041.637,E2 -15041.637} C_VEL
LIN {X 0,Y 370.284,Z 137.602,A -85,B 0,C 180,E1 -15043.165,E2 -15043.165} C_VEL
LIN {X 0,Y 368.086,Z 135.567,A -85,B 0,C 180,E1 -15043.933,E2 -15043.933} C_VEL
LIN {X 0,Y 363.708,Z 131.956,A -85,B 0,C 180,E1 -15045.342,E2 -15045.342} C_VEL
LIN {X 0,Y 360.456,Z 128.551,A -85,B 0,C 180,E1 -15046.335,E2 -15046.335} C_VEL
LIN {X 0,Y 356.255,Z 124.937,A -85,B 0,C 180,E1 -15047.492,E2 -15047.492} C_VEL
LIN {X 0,Y 353.161,Z 121.708,A -85,B 0,C 180,E1 -15048.309,E2 -15048.309} C_VEL
LIN {X 0,Y 349.304,Z 117.883,A -85,B 0,C 180,E1 -15049.285,E2 -15049.285} C_VEL
LIN {X 0,Y 346.781,Z 115.105,A -85,B 0,C 180,E1 -15049.881,E2 -15049.881} C_VEL
LIN {X 0,Y 343.085,Z 111.04,A -85,B 0,C 180,E1 -15050.756,E2 -15050.756} C_VEL
LIN {X 0,Y 338.395,Z 105.801,A -85,B 0,C 180,E1 -15051.78,E2 -15051.78} C_VEL
LIN {X 0,Y 336.612,Z 103.599,A -85,B 0,C 180,E1 -15052.177,E2 -15052.177} C_VEL
LIN {X 0,Y 333.567,Z 99.716,A -85,B 0,C 180,E1 -15052.804,E2 -15052.804} C_VEL
LIN {X 0,Y 330.474,Z 95.835,A -85,B 0,C 180,E1 -15053.45,E2 -15053.45} C_VEL
LIN {X 0,Y 329.168,Z 93.914,A -85,B 0,C 180,E1 -15053.716,E2 -15053.716} C_VEL
LIN {X 0,Y 327.269,Z 91.475,A -85,B 0,C 180,E1 -15054.08,E2 -15054.08} C_VEL
LIN {X 0,Y 326.718,Z 89.741,A -85,B 0,C 180,E1 -15054.335,E2 -15054.335} C_VEL
LIN {X 0,Y 326.685,Z 89.294,A -85,B 0,C 180,E1 -15054.803,E2 -15054.803} C_VEL
LIN {X 0,Y 326.646,Z 89.282,A -85,B 0,C 180,E1 -15058.251,E2 -15058.251} C_VEL
LIN {X 0,Y 326.587,Z 89.302,A -85,B 0,C 180,E1 -15061.096,E2 -15061.096} C_VEL
LIN {X 0,Y 326.603,Z 89.271,A -85,B 0,C 180,E1 -15064.02,E2 -15064.02} C_VEL
LIN {X 0,Y 326.624,Z 89.297,A -85,B 0,C 180,E1 -15067.239,E2 -15067.239} C_VEL
LIN {X 0,Y 326.573,Z 89.262,A -85,B 0,C 180,E1 -15071.132,E2 -15071.132} C_VEL
LIN {X 0,Y 326.525,Z 89.299,A -85,B 0,C 180,E1 -15074.743,E2 -15074.743} C_VEL
LIN {X 0,Y 326.592,Z 89.296,A -85,B 0,C 180,E1 -15078.158,E2 -15078.158} C_VEL
LIN {X 0,Y 326.64,Z 89.296,A -85,B 0,C 180,E1 -15081.395,E2 -15081.395} C_VEL
LIN {X 0,Y 326.617,Z 89.284,A -85,B 0,C 180,E1 -15084.852,E2 -15084.852} C_VEL
LIN {X 0,Y 326.605,Z 89.297,A -85,B 0,C 180,E1 -15087.456,E2 -15087.456} C_VEL
LIN {X 0,Y 326.645,Z 89.295,A -85,B 0,C 180,E1 -15090.34,E2 -15090.34} C_VEL
LIN {X 0,Y 326.688,Z 89.279,A -85,B 0,C 180,E1 -15094.517,E2 -15094.517} C_VEL
LIN {X 0,Y 326.644,Z 89.288,A -85,B 0,C 180,E1 -15098.546,E2 -15098.546} C_VEL
LIN {X 0,Y 326.743,Z 89.255,A -85,B 0,C 180,E1 -15101.178,E2 -15101.178} C_VEL
LIN {X 0,Y 326.756,Z 89.282,A -85,B 0,C 180,E1 -15105.272,E2 -15105.272} C_VEL
LIN {X 0,Y 326.106,Z 89.364,A -85,B 0,C 180,E1 -15106.301,E2 -15106.301} C_VEL
LIN {X 0,Y 323.242,Z 89.706,A -85,B 0,C 180,E1 -15107.976,E2 -15107.976} C_VEL
LIN {X 0,Y 320.836,Z 89.991,A -85,B 0,C 180,E1 -15109.333,E2 -15109.333} C_VEL
LIN {X 0,Y 319.851,Z 90.109,A -85,B 0,C 180,E1 -15110.383,E2 -15110.383} C_VEL
LIN {X 0,Y 319.797,Z 90.117,A -85,B 0,C 180,E1 -15110.739,E2 -15110.739} C_VEL
LIN {X 0,Y 319.951,Z 90.125,A -85,B 0,C 180,E1 -15113.695,E2 -15113.695} C_VEL
LIN {X 0,Y 319.989,Z 90.113,A -85,B 0,C 180,E1 -15117.483,E2 -15117.483} C_VEL
LIN {X 0,Y 320.131,Z 90.073,A -85,B 0,C 180,E1 -15120.001,E2 -15120.001} C_VEL
LIN {X 0,Y 319.99,Z 90.115,A -85,B 0,C 180,E1 -15122.518,E2 -15122.518} C_VEL
LIN {X 0,Y 319.954,Z 90.124,A -85,B 0,C 180,E1 -15126.306,E2 -15126.306} C_VEL
LIN {X 0,Y 319.843,Z 90.113,A -85,B 0,C 180,E1 -15128.849,E2 -15128.849} C_VEL
LIN {X 0,Y 319.682,Z 90.155,A -85,B 0,C 180,E1 -15132.7,E2 -15132.7} C_VEL
LIN {X 0,Y 319.7,Z 90.159,A -85,B 0,C 180,E1 -15135.296,E2 -15135.296} C_VEL
LIN {X 0,Y 319.675,Z 90.132,A -85,B 0,C 180,E1 -15139.256,E2 -15139.256} C_VEL
LIN {X 0,Y 319.572,Z 90.178,A -85,B 0,C 180,E1 -15143.32,E2 -15143.32} C_VEL
LIN {X 0,Y 319.635,Z 90.149,A -85,B 0,C 180,E1 -15146.089,E2 -15146.089} C_VEL
LIN {X 0,Y 319.581,Z 90.165,A -85,B 0,C 180,E1 -15148.935,E2 -15148.935} C_VEL
LIN {X 0,Y 319.532,Z 90.179,A -85,B 0,C 180,E1 -15151.863,E2 -15151.863} C_VEL
LIN {X 0,Y 319.581,Z 90.166,A -85,B 0,C 180,E1 -15155.544,E2 -15155.544} C_VEL
LIN {X 0,Y 319.558,Z 90.178,A -85,B 0,C 180,E1 -15158.011,E2 -15158.011} C_VEL
LIN {X 0,Y 319.527,Z 90.181,A -85,B 0,C 180,E1 -15161.598,E2 -15161.598} C_VEL
LIN {X 0,Y 319.49,Z 90.18,A -85,B 0,C 180,E1 -15165.258,E2 -15165.258} C_VEL
LIN {X 0,Y 319.53,Z 90.162,A -85,B 0,C 180,E1 -15168.712,E2 -15168.712} C_VEL
LIN {X 0,Y 319.581,Z 90.178,A -85,B 0,C 180,E1 -15172.344,E2 -15172.344} C_VEL
LIN {X 0,Y 319.633,Z 90.375,A -85,B 0,C 180,E1 -15176.106,E2 -15176.106} C_VEL
LIN {X 0,Y 320.923,Z 96.75,A -85,B 0,C 180,E1 -15178.659,E2 -15178.659} C_VEL
LIN {X 0,Y 322.739,Z 105.867,A -85,B 0,C 180,E1 -15182.084,E2 -15182.084} C_VEL
LIN {X 0,Y 323.043,Z 110.186,A -85,B 0,C 180,E1 -15183.661,E2 -15183.661} C_VEL
LIN {X 0,Y 322.585,Z 113.845,A -85,B 0,C 180,E1 -15184.85,E2 -15184.85} C_VEL
LIN {X 0,Y 324.639,Z 123.261,A -85,B 0,C 180,E1 -15185.293,E2 -15185.293} C_VEL
LIN {X 0,Y 328.95,Z 144.879,A -85,B 0,C 180,E1 -15186.14,E2 -15186.14} C_VEL
LIN {X 0,Y 330.565,Z 155.098,A -85,B 0,C 180,E1 -15186.5,E2 -15186.5} C_VEL
LIN {X 0,Y 329.247,Z 218.575,A -85,B 0,C 180,E1 -15187.901,E2 -15187.901} C_VEL
LIN {X 0,Y 328.672,Z 229.299,A -85,B 0,C 180,E1 -15188.273,E2 -15188.273} C_VEL
LIN {X 0,Y 327.942,Z 238.397,A -85,B 0,C 180,E1 -15188.717,E2 -15188.717} C_VEL
LIN {X 0,Y 327.106,Z 247.752,A -85,B 0,C 180,E1 -15189.319,E2 -15189.319} C_VEL
LIN {X 0,Y 325.993,Z 257.891,A -85,B 0,C 180,E1 -15190.151,E2 -15190.151} C_VEL
LIN {X 0,Y 324.852,Z 266.885,A -85,B 0,C 180,E1 -15191.064,E2 -15191.064} C_VEL
LIN {X 0,Y 323.69,Z 275.612,A -85,B 0,C 180,E1 -15192.141,E2 -15192.141} C_VEL
LIN {X 0,Y 322.641,Z 283.005,A -85,B 0,C 180,E1 -15193.225,E2 -15193.225} C_VEL
LIN {X 0,Y 321.628,Z 290.598,A -85,B 0,C 180,E1 -15194.548,E2 -15194.548} C_VEL
LIN {X 0,Y 320.614,Z 297.805,A -85,B 0,C 180,E1 -15196.047,E2 -15196.047} C_VEL
LIN {X 0,Y 319.624,Z 304.12,A -85,B 0,C 180,E1 -15197.621,E2 -15197.621} C_VEL
LIN {X 0,Y 318.936,Z 309.383,A -85,B 0,C 180,E1 -15199.205,E2 -15199.205} C_VEL
LIN {X 0,Y 318.36,Z 314.514,A -85,B 0,C 180,E1 -15201.111,E2 -15201.111} C_VEL
LIN {X 0,Y 317.991,Z 318.503,A -85,B 0,C 180,E1 -15203.018,E2 -15203.018} C_VEL
LIN {X 0,Y 317.8,Z 321.453,A -85,B 0,C 180,E1 -15204.925,E2 -15204.925} C_VEL
LIN {X 0,Y 317.756,Z 323.901,A -85,B 0,C 180,E1 -15207.465,E2 -15207.465} C_VEL
LIN {X 0,Y 317.734,Z 324.49,A -85,B 0,C 180,E1 -15208.733,E2 -15208.733} C_VEL
LIN {X 0,Y 317.734,Z 324.49,A -85,B 0,C 180,E1 -15211.267,E2 -15211.267} C_VEL
LIN {X 0,Y 317.756,Z 323.901,A -85,B 0,C 180,E1 -15212.535,E2 -15212.535} C_VEL
LIN {X 0,Y 317.795,Z 321.453,A -85,B 0,C 180,E1 -15215.075,E2 -15215.075} C_VEL
LIN {X 0,Y 317.987,Z 318.503,A -85,B 0,C 180,E1 -15216.982,E2 -15216.982} C_VEL
LIN {X 0,Y 318.36,Z 314.514,A -85,B 0,C 180,E1 -15218.889,E2 -15218.889} C_VEL
LIN {X 0,Y 318.935,Z 309.383,A -85,B 0,C 180,E1 -15220.795,E2 -15220.795} C_VEL
LIN {X 0,Y 319.616,Z 304.119,A -85,B 0,C 180,E1 -15222.38,E2 -15222.38} C_VEL
LIN {X 0,Y 320.615,Z 297.805,A -85,B 0,C 180,E1 -15223.953,E2 -15223.953} C_VEL
LIN {X 0,Y 321.441,Z 291.853,A -85,B 0,C 180,E1 -15225.211,E2 -15225.211} C_VEL
LIN {X 0,Y 322.41,Z 284.926,A -85,B 0,C 180,E1 -15226.462,E2 -15226.462} C_VEL
LIN {X 0,Y 323.538,Z 276.746,A -85,B 0,C 180,E1 -15227.705,E2 -15227.705} C_VEL
LIN {X 0,Y 324.707,Z 268.237,A -85,B 0,C 180,E1 -15228.781,E2 -15228.781} C_VEL
LIN {X 0,Y 325.847,Z 259.524,A -85,B 0,C 180,E1 -15229.695,E2 -15229.695} C_VEL
LIN {X 0,Y 326.923,Z 249.767,A -85,B 0,C 180,E1 -15230.529,E2 -15230.529} C_VEL
LIN {X 0,Y 327.765,Z 240.974,A -85,B 0,C 180,E1 -15231.131,E2 -15231.131} C_VEL
LIN {X 0,Y 328.556,Z 231.047,A -85,B 0,C 180,E1 -15231.653,E2 -15231.653} C_VEL
LIN {X 0,Y 329.073,Z 221.19,A -85,B 0,C 180,E1 -15232.029,E2 -15232.029} C_VEL
LIN {X 0,Y 329.718,Z 198.37,A -85,B 0,C 180,E1 -15232.561,E2 -15232.561} C_VEL
LIN {X 0,Y 330.534,Z 154.474,A -85,B 0,C 180,E1 -15233.517,E2 -15233.517} C_VEL
LIN {X 0,Y 326.235,Z 130.689,A -85,B 0,C 180,E1 -15234.404,E2 -15234.404} C_VEL
LIN {X 0,Y 322.602,Z 114.009,A -85,B 0,C 180,E1 -15235.129,E2 -15235.129} C_VEL
LIN {X 0,Y 322.692,Z 112.54,A -85,B 0,C 180,E1 -15235.511,E2 -15235.511} C_VEL
LIN {X 0,Y 323.092,Z 108.643,A -85,B 0,C 180,E1 -15236.893,E2 -15236.893} C_VEL
LIN {X 0,Y 321.9,Z 101.414,A -85,B 0,C 180,E1 -15239.601,E2 -15239.601} C_VEL
LIN {X 0,Y 320.159,Z 92.816,A -85,B 0,C 180,E1 -15242.909,E2 -15242.909} C_VEL
LIN {X 0,Y 319.586,Z 90.195,A -85,B 0,C 180,E1 -15244.013,E2 -15244.013} C_VEL
LIN {X 0,Y 319.576,Z 90.175,A -85,B 0,C 180,E1 -15248.007,E2 -15248.007} C_VEL
LIN {X 0,Y 319.527,Z 90.167,A -85,B 0,C 180,E1 -15251.596,E2 -15251.596} C_VEL
LIN {X 0,Y 319.49,Z 90.18,A -85,B 0,C 180,E1 -15255.257,E2 -15255.257} C_VEL
LIN {X 0,Y 319.53,Z 90.177,A -85,B 0,C 180,E1 -15258.711,E2 -15258.711} C_VEL
LIN {X 0,Y 319.563,Z 90.178,A -85,B 0,C 180,E1 -15262.347,E2 -15262.347} C_VEL
LIN {X 0,Y 319.561,Z 90.16,A -85,B 0,C 180,E1 -15265.123,E2 -15265.123} C_VEL
LIN {X 0,Y 319.567,Z 90.181,A -85,B 0,C 180,E1 -15269.059,E2 -15269.059} C_VEL
LIN {X 0,Y 319.606,Z 90.149,A -85,B 0,C 180,E1 -15272.497,E2 -15272.497} C_VEL
LIN {X 0,Y 319.607,Z 90.167,A -85,B 0,C 180,E1 -15275.303,E2 -15275.303} C_VEL
LIN {X 0,Y 319.598,Z 90.171,A -85,B 0,C 180,E1 -15278.047,E2 -15278.047} C_VEL
LIN {X 0,Y 319.69,Z 90.13,A -85,B 0,C 180,E1 -15280.962,E2 -15280.962} C_VEL
LIN {X 0,Y 319.732,Z 90.154,A -85,B 0,C 180,E1 -15285.275,E2 -15285.275} C_VEL
LIN {X 0,Y 319.758,Z 90.12,A -85,B 0,C 180,E1 -15289.872,E2 -15289.872} C_VEL
LIN {X 0,Y 319.935,Z 90.115,A -85,B 0,C 180,E1 -15292.426,E2 -15292.426} C_VEL
LIN {X 0,Y 319.748,Z 90.154,A -85,B 0,C 180,E1 -15294.955,E2 -15294.955} C_VEL
LIN {X 0,Y 319.99,Z 90.115,A -85,B 0,C 180,E1 -15297.482,E2 -15297.482} C_VEL
LIN {X 0,Y 320.131,Z 90.073,A -85,B 0,C 180,E1 -15299.999,E2 -15299.999} C_VEL
LIN {X 0,Y 319.989,Z 90.113,A -85,B 0,C 180,E1 -15302.517,E2 -15302.517} C_VEL
LIN {X 0,Y 319.931,Z 90.123,A -85,B 0,C 180,E1 -15306.644,E2 -15306.644} C_VEL
LIN {X 0,Y 319.758,Z 90.121,A -85,B 0,C 180,E1 -15310.126,E2 -15310.126} C_VEL
LIN {X 0,Y 319.73,Z 90.157,A -85,B 0,C 180,E1 -15314.724,E2 -15314.724} C_VEL
LIN {X 0,Y 319.687,Z 90.133,A -85,B 0,C 180,E1 -15319.037,E2 -15319.037} C_VEL
LIN {X 0,Y 319.569,Z 90.18,A -85,B 0,C 180,E1 -15323.319,E2 -15323.319} C_VEL
LIN {X 0,Y 319.632,Z 90.154,A -85,B 0,C 180,E1 -15326.087,E2 -15326.087} C_VEL
LIN {X 0,Y 319.577,Z 90.164,A -85,B 0,C 180,E1 -15328.934,E2 -15328.934} C_VEL
LIN {X 0,Y 319.528,Z 90.182,A -85,B 0,C 180,E1 -15331.861,E2 -15331.861} C_VEL
LIN {X 0,Y 319.577,Z 90.165,A -85,B 0,C 180,E1 -15335.543,E2 -15335.543} C_VEL
LIN {X 0,Y 319.579,Z 90.178,A -85,B 0,C 180,E1 -15338.006,E2 -15338.006} C_VEL
LIN {X 0,Y 319.563,Z 90.17,A -85,B 0,C 180,E1 -15341.605,E2 -15341.605} C_VEL
LIN {X 0,Y 319.486,Z 90.175,A -85,B 0,C 180,E1 -15345.257,E2 -15345.257} C_VEL
LIN {X 0,Y 319.524,Z 90.138,A -85,B 0,C 180,E1 -15348.711,E2 -15348.711} C_VEL
LIN {X 0,Y 319.574,Z 90.179,A -85,B 0,C 180,E1 -15352.344,E2 -15352.344} C_VEL
LIN {X 0,Y 319.556,Z 90.147,A -85,B 0,C 180,E1 -15355.123,E2 -15355.123} C_VEL
LIN {X 0,Y 319.563,Z 90.172,A -85,B 0,C 180,E1 -15359.059,E2 -15359.059} C_VEL
LIN {X 0,Y 319.602,Z 90.171,A -85,B 0,C 180,E1 -15362.498,E2 -15362.498} C_VEL
LIN {X 0,Y 319.676,Z 90.391,A -85,B 0,C 180,E1 -15364.614,E2 -15364.614} C_VEL
LIN {X 0,Y 319.92,Z 91.454,A -85,B 0,C 180,E1 -15364.853,E2 -15364.853} C_VEL
LIN {X 0,Y 321.679,Z 94.338,A -85,B 0,C 180,E1 -15365.191,E2 -15365.191} C_VEL
LIN {X 0,Y 324.766,Z 98.844,A -85,B 0,C 180,E1 -15365.751,E2 -15365.751} C_VEL
LIN {X 0,Y 326.817,Z 101.576,A -85,B 0,C 180,E1 -15366.145,E2 -15366.145} C_VEL
LIN {X 0,Y 330.677,Z 106.375,A -85,B 0,C 180,E1 -15366.898,E2 -15366.898} C_VEL
LIN {X 0,Y 337.761,Z 114.697,A -85,B 0,C 180,E1 -15368.376,E2 -15368.376} C_VEL
LIN {X 0,Y 340.438,Z 117.599,A -85,B 0,C 180,E1 -15368.958,E2 -15368.958} C_VEL
LIN {X 0,Y 344.628,Z 121.859,A -85,B 0,C 180,E1 -15369.9,E2 -15369.9} C_VEL
LIN {X 0,Y 349.572,Z 127.111,A -85,B 0,C 180,E1 -15371.08,E2 -15371.08} C_VEL
LIN {X 0,Y 352.228,Z 129.568,A -85,B 0,C 180,E1 -15371.748,E2 -15371.748} C_VEL
LIN {X 0,Y 356.691,Z 133.888,A -85,B 0,C 180,E1 -15372.934,E2 -15372.934} C_VEL
LIN {X 0,Y 359.645,Z 136.335,A -85,B 0,C 180,E1 -15373.746,E2 -15373.746} C_VEL
LIN {X 0,Y 364,Z 140.521,A -85,B 0,C 180,E1 -15375.073,E2 -15375.073} C_VEL
LIN {X 0,Y 367.974,Z 143.699,A -85,B 0,C 180,E1 -15376.368,E2 -15376.368} C_VEL
LIN {X 0,Y 372.205,Z 147.583,A -85,B 0,C 180,E1 -15377.936,E2 -15377.936} C_VEL
LIN {X 0,Y 376.1,Z 150.109,A -85,B 0,C 180,E1 -15379.54,E2 -15379.54} C_VEL
LIN {X 0,Y 377.407,Z 151.142,A -85,B 0,C 180,E1 -15380.169,E2 -15380.169} C_VEL
LIN {X 0,Y 380.163,Z 153.983,A -85,B 0,C 180,E1 -15381.649,E2 -15381.649} C_VEL
LIN {X 0,Y 382.58,Z 155.842,A -85,B 0,C 180,E1 -15383.16,E2 -15383.16} C_VEL
LIN {X 0,Y 384.638,Z 157.028,A -85,B 0,C 180,E1 -15384.758,E2 -15384.758} C_VEL
LIN {X 0,Y 386.062,Z 157.612,A -85,B 0,C 180,E1 -15386.193,E2 -15386.193} C_VEL
LIN {X 0,Y 387.31,Z 158.161,A -85,B 0,C 180,E1 -15388.199,E2 -15388.199} C_VEL
LIN {X 0,Y 387.677,Z 158.274,A -85,B 0,C 180,E1 -15390,E2 -15390} C_VEL
LIN {X 0,Y 387.389,Z 158.231,A -85,B 0,C 180,E1 -15391.559,E2 -15391.559} C_VEL
LIN {X 0,Y 386.606,Z 157.789,A -85,B 0,C 180,E1 -15393.126,E2 -15393.126} C_VEL
LIN {X 0,Y 384.954,Z 157.186,A -85,B 0,C 180,E1 -15394.966,E2 -15394.966} C_VEL
LIN {X 0,Y 382.89,Z 156.034,A -85,B 0,C 180,E1 -15396.624,E2 -15396.624} C_VEL
LIN {X 0,Y 380.324,Z 154.132,A -85,B 0,C 180,E1 -15398.255,E2 -15398.255} C_VEL
LIN {X 0,Y 377.464,Z 151.225,A -85,B 0,C 180,E1 -15399.8,E2 -15399.8} C_VEL
LIN {X 0,Y 376.153,Z 150.137,A -85,B 0,C 180,E1 -15400.437,E2 -15400.437} C_VEL
LIN {X 0,Y 372.208,Z 147.589,A -85,B 0,C 180,E1 -15402.063,E2 -15402.063} C_VEL
LIN {X 0,Y 368.208,Z 143.92,A -85,B 0,C 180,E1 -15403.553,E2 -15403.553} C_VEL
LIN {X 0,Y 365.754,Z 141.855,A -85,B 0,C 180,E1 -15404.37,E2 -15404.37} C_VEL
LIN {X 0,Y 361.306,Z 138.142,A -85,B 0,C 180,E1 -15405.748,E2 -15405.748} C_VEL
LIN {X 0,Y 358.078,Z 134.925,A -85,B 0,C 180,E1 -15406.696,E2 -15406.696} C_VEL
LIN {X 0,Y 353.582,Z 130.99,A -85,B 0,C 180,E1 -15407.907,E2 -15407.907} C_VEL
LIN {X 0,Y 350.586,Z 127.955,A -85,B 0,C 180,E1 -15408.666,E2 -15408.666} C_VEL
LIN {X 0,Y 346.501,Z 124.028,A -85,B 0,C 180,E1 -15409.655,E2 -15409.655} C_VEL
LIN {X 0,Y 343.552,Z 120.879,A -85,B 0,C 180,E1 -15410.351,E2 -15410.351} C_VEL
LIN {X 0,Y 339.504,Z 116.425,A -85,B 0,C 180,E1 -15411.248,E2 -15411.248} C_VEL
LIN {X 0,Y 335.087,Z 111.617,A -85,B 0,C 180,E1 -15412.201,E2 -15412.201} C_VEL
LIN {X 0,Y 329.948,Z 105.266,A -85,B 0,C 180,E1 -15413.26,E2 -15413.26} C_VEL
LIN {X 0,Y 326.373,Z 100.922,A -85,B 0,C 180,E1 -15413.942,E2 -15413.942} C_VEL
LIN {X 0,Y 324.773,Z 98.849,A -85,B 0,C 180,E1 -15414.248,E2 -15414.248} C_VEL
LIN {X 0,Y 322.407,Z 95.359,A -85,B 0,C 180,E1 -15414.685,E2 -15414.685} C_VEL
LIN {X 0,Y 320.021,Z 91.733,A -85,B 0,C 180,E1 -15415.124,E2 -15415.124} C_VEL
LIN {X 0,Y 319.702,Z 90.479,A -85,B 0,C 180,E1 -15415.339,E2 -15415.339} C_VEL
LIN {X 0,Y 319.63,Z 90.172,A -85,B 0,C 180,E1 -15416.088,E2 -15416.088} C_VEL
LIN {X 0,Y 319.576,Z 90.156,A -85,B 0,C 180,E1 -15418.935,E2 -15418.935} C_VEL
LIN {X 0,Y 319.527,Z 90.186,A -85,B 0,C 180,E1 -15421.862,E2 -15421.862} C_VEL
LIN {X 0,Y 319.576,Z 90.147,A -85,B 0,C 180,E1 -15425.543,E2 -15425.543} C_VEL
LIN {X 0,Y 319.569,Z 90.181,A -85,B 0,C 180,E1 -15428.008,E2 -15428.008} C_VEL
LIN {X 0,Y 319.522,Z 90.135,A -85,B 0,C 180,E1 -15431.597,E2 -15431.597} C_VEL
LIN {X 0,Y 319.487,Z 90.18,A -85,B 0,C 180,E1 -15435.258,E2 -15435.258} C_VEL
LIN {X 0,Y 319.539,Z 90.169,A -85,B 0,C 180,E1 -15438.715,E2 -15438.715} C_VEL
LIN {X 0,Y 319.579,Z 90.177,A -85,B 0,C 180,E1 -15442.344,E2 -15442.344} C_VEL
LIN {X 0,Y 319.557,Z 90.161,A -85,B 0,C 180,E1 -15445.124,E2 -15445.124} C_VEL
LIN {X 0,Y 319.564,Z 90.182,A -85,B 0,C 180,E1 -15449.06,E2 -15449.06} C_VEL
LIN {X 0,Y 319.603,Z 90.15,A -85,B 0,C 180,E1 -15452.498,E2 -15452.498} C_VEL
LIN {X 0,Y 319.603,Z 90.171,A -85,B 0,C 180,E1 -15455.305,E2 -15455.305} C_VEL
LIN {X 0,Y 319.595,Z 90.172,A -85,B 0,C 180,E1 -15458.048,E2 -15458.048} C_VEL
LIN {X 0,Y 319.687,Z 90.133,A -85,B 0,C 180,E1 -15460.963,E2 -15460.963} C_VEL
LIN {X 0,Y 319.73,Z 90.157,A -85,B 0,C 180,E1 -15465.276,E2 -15465.276} C_VEL
LIN {X 0,Y 319.758,Z 90.121,A -85,B 0,C 180,E1 -15469.874,E2 -15469.874} C_VEL
LIN {X 0,Y 319.797,Z 90.117,A -85,B 0,C 180,E1 -15470.739,E2 -15470.739} C_VEL
LIN {X 0,Y 319.52,Z 90.159,A -85,B 0,C 180,E1 -15471.443,E2 -15471.443} C_VEL
LIN {X 0,Y 318.158,Z 90.34,A -85,B 0,C 180,E1 -15472.479,E2 -15472.479} C_VEL
LIN {X 0,Y 313.746,Z 90.906,A -85,B 0,C 180,E1 -15474.886,E2 -15474.886} C_VEL
LIN {X 0,Y 312.756,Z 91.026,A -85,B 0,C 180,E1 -15475.961,E2 -15475.961} C_VEL
LIN {X 0,Y 312.718,Z 91.026,A -85,B 0,C 180,E1 -15476.325,E2 -15476.325} C_VEL
LIN {X 0,Y 312.988,Z 90.97,A -85,B 0,C 180,E1 -15478.714,E2 -15478.714} C_VEL
LIN {X 0,Y 312.988,Z 90.972,A -85,B 0,C 180,E1 -15481.287,E2 -15481.287} C_VEL
LIN {X 0,Y 312.719,Z 91.03,A -85,B 0,C 180,E1 -15485.158,E2 -15485.158} C_VEL
LIN {X 0,Y 312.873,Z 90.992,A -85,B 0,C 180,E1 -15487.746,E2 -15487.746} C_VEL
LIN {X 0,Y 312.67,Z 91.017,A -85,B 0,C 180,E1 -15491.672,E2 -15491.672} C_VEL
LIN {X 0,Y 312.701,Z 91.03,A -85,B 0,C 180,E1 -15494.888,E2 -15494.888} C_VEL
LIN {X 0,Y 312.631,Z 91.009,A -85,B 0,C 180,E1 -15499.237,E2 -15499.237} C_VEL
LIN {X 0,Y 312.547,Z 91.05,A -85,B 0,C 180,E1 -15502.79,E2 -15502.79} C_VEL
LIN {X 0,Y 312.603,Z 91.026,A -85,B 0,C 180,E1 -15505.936,E2 -15505.936} C_VEL
LIN {X 0,Y 312.539,Z 91.052,A -85,B 0,C 180,E1 -15509.651,E2 -15509.651} C_VEL
LIN {X 0,Y 312.521,Z 91.036,A -85,B 0,C 180,E1 -15513.689,E2 -15513.689} C_VEL
LIN {X 0,Y 312.527,Z 91.055,A -85,B 0,C 180,E1 -15517.386,E2 -15517.386} C_VEL
LIN {X 0,Y 312.492,Z 91.047,A -85,B 0,C 180,E1 -15520.71,E2 -15520.71} C_VEL
LIN {X 0,Y 312.453,Z 91.057,A -85,B 0,C 180,E1 -15524.21,E2 -15524.21} C_VEL
LIN {X 0,Y 312.486,Z 91.051,A -85,B 0,C 180,E1 -15527.919,E2 -15527.919} C_VEL
LIN {X 0,Y 312.538,Z 91.049,A -85,B 0,C 180,E1 -15531.911,E2 -15531.911} C_VEL
LIN {X 0,Y 312.561,Z 91.164,A -85,B 0,C 180,E1 -15535.602,E2 -15535.602} C_VEL
LIN {X 0,Y 313.928,Z 97.712,A -85,B 0,C 180,E1 -15538.291,E2 -15538.291} C_VEL
LIN {X 0,Y 315.505,Z 105.662,A -85,B 0,C 180,E1 -15541.385,E2 -15541.385} C_VEL
LIN {X 0,Y 316.097,Z 110.444,A -85,B 0,C 180,E1 -15543.204,E2 -15543.204} C_VEL
LIN {X 0,Y 315.812,Z 113.53,A -85,B 0,C 180,E1 -15544.252,E2 -15544.252} C_VEL
LIN {X 0,Y 316.767,Z 118.082,A -85,B 0,C 180,E1 -15544.514,E2 -15544.514} C_VEL
LIN {X 0,Y 321.365,Z 139.936,A -85,B 0,C 180,E1 -15545.427,E2 -15545.427} C_VEL
LIN {X 0,Y 324.052,Z 156.055,A -85,B 0,C 180,E1 -15546.026,E2 -15546.026} C_VEL
LIN {X 0,Y 322.688,Z 218.391,A -85,B 0,C 180,E1 -15547.427,E2 -15547.427} C_VEL
LIN {X 0,Y 322.091,Z 229.108,A -85,B 0,C 180,E1 -15547.805,E2 -15547.805} C_VEL
LIN {X 0,Y 321.341,Z 238.207,A -85,B 0,C 180,E1 -15548.258,E2 -15548.258} C_VEL
LIN {X 0,Y 320.364,Z 248.568,A -85,B 0,C 180,E1 -15548.947,E2 -15548.947} C_VEL
LIN {X 0,Y 319.305,Z 257.7,A -85,B 0,C 180,E1 -15549.717,E2 -15549.717} C_VEL
LIN {X 0,Y 318.131,Z 266.694,A -85,B 0,C 180,E1 -15550.648,E2 -15550.648} C_VEL
LIN {X 0,Y 316.932,Z 275.421,A -85,B 0,C 180,E1 -15551.746,E2 -15551.746} C_VEL
LIN {X 0,Y 315.815,Z 282.814,A -85,B 0,C 180,E1 -15552.851,E2 -15552.851} C_VEL
LIN {X 0,Y 314.748,Z 290.573,A -85,B 0,C 180,E1 -15554.235,E2 -15554.235} C_VEL
LIN {X 0,Y 313.692,Z 297.614,A -85,B 0,C 180,E1 -15555.733,E2 -15555.733} C_VEL
LIN {X 0,Y 312.667,Z 303.928,A -85,B 0,C 180,E1 -15557.341,E2 -15557.341} C_VEL
LIN {X 0,Y 311.934,Z 309.191,A -85,B 0,C 180,E1 -15558.959,E2 -15558.959} C_VEL
LIN {X 0,Y 311.306,Z 314.322,A -85,B 0,C 180,E1 -15560.907,E2 -15560.907} C_VEL
LIN {X 0,Y 310.922,Z 318.312,A -85,B 0,C 180,E1 -15562.859,E2 -15562.859} C_VEL
LIN {X 0,Y 310.704,Z 321.262,A -85,B 0,C 180,E1 -15564.809,E2 -15564.809} C_VEL
LIN {X 0,Y 310.679,Z 323.711,A -85,B 0,C 180,E1 -15567.407,E2 -15567.407} C_VEL
LIN {X 0,Y 310.649,Z 324.3,A -85,B 0,C 180,E1 -15568.704,E2 -15568.704} C_VEL
LIN {X 0,Y 310.649,Z 324.3,A -85,B 0,C 180,E1 -15571.296,E2 -15571.296} C_VEL
LIN {X 0,Y 310.679,Z 323.711,A -85,B 0,C 180,E1 -15572.593,E2 -15572.593} C_VEL
LIN {X 0,Y 310.699,Z 321.262,A -85,B 0,C 180,E1 -15575.191,E2 -15575.191} C_VEL
LIN {X 0,Y 310.919,Z 318.312,A -85,B 0,C 180,E1 -15577.142,E2 -15577.142} C_VEL
LIN {X 0,Y 311.306,Z 314.322,A -85,B 0,C 180,E1 -15579.093,E2 -15579.093} C_VEL
LIN {X 0,Y 311.934,Z 309.191,A -85,B 0,C 180,E1 -15581.041,E2 -15581.041} C_VEL
LIN {X 0,Y 312.66,Z 303.928,A -85,B 0,C 180,E1 -15582.66,E2 -15582.66} C_VEL
LIN {X 0,Y 313.702,Z 297.614,A -85,B 0,C 180,E1 -15584.267,E2 -15584.267} C_VEL
LIN {X 0,Y 314.805,Z 290.449,A -85,B 0,C 180,E1 -15585.787,E2 -15585.787} C_VEL
LIN {X 0,Y 315.897,Z 282.816,A -85,B 0,C 180,E1 -15587.144,E2 -15587.144} C_VEL
LIN {X 0,Y 317.114,Z 274.287,A -85,B 0,C 180,E1 -15588.41,E2 -15588.41} C_VEL
LIN {X 0,Y 318.561,Z 263.993,A -85,B 0,C 180,E1 -15589.66,E2 -15589.66} C_VEL
LIN {X 0,Y 320.024,Z 251.588,A -85,B 0,C 180,E1 -15590.823,E2 -15590.823} C_VEL
LIN {X 0,Y 321.145,Z 240.783,A -85,B 0,C 180,E1 -15591.588,E2 -15591.588} C_VEL
LIN {X 0,Y 321.982,Z 230.857,A -85,B 0,C 180,E1 -15592.118,E2 -15592.118} C_VEL
LIN {X 0,Y 322.503,Z 221,A -85,B 0,C 180,E1 -15592.502,E2 -15592.502} C_VEL
LIN {X 0,Y 323.174,Z 198.179,A -85,B 0,C 180,E1 -15593.044,E2 -15593.044} C_VEL
LIN {X 0,Y 324.047,Z 155.458,A -85,B 0,C 180,E1 -15593.989,E2 -15593.989} C_VEL
LIN {X 0,Y 319.668,Z 131.346,A -85,B 0,C 180,E1 -15594.918,E2 -15594.918} C_VEL
LIN {X 0,Y 315.82,Z 113.872,A -85,B 0,C 180,E1 -15595.702,E2 -15595.702} C_VEL
LIN {X 0,Y 315.92,Z 112.442,A -85,B 0,C 180,E1 -15596.063,E2 -15596.063} C_VEL
LIN {X 0,Y 316.082,Z 109.351,A -85,B 0,C 180,E1 -15597.202,E2 -15597.202} C_VEL
LIN {X 0,Y 314.751,Z 101.701,A -85,B 0,C 180,E1 -15600.158,E2 -15600.158} C_VEL
LIN {X 0,Y 313.203,Z 94.133,A -85,B 0,C 180,E1 -15603.158,E2 -15603.158} C_VEL
LIN {X 0,Y 312.531,Z 91.073,A -85,B 0,C 180,E1 -15604.499,E2 -15604.499} C_VEL
LIN {X 0,Y 312.538,Z 91.05,A -85,B 0,C 180,E1 -15608.089,E2 -15608.089} C_VEL
LIN {X 0,Y 312.486,Z 91.051,A -85,B 0,C 180,E1 -15612.081,E2 -15612.081} C_VEL
LIN {X 0,Y 312.46,Z 91.06,A -85,B 0,C 180,E1 -15616.034,E2 -15616.034} C_VEL
LIN {X 0,Y 312.506,Z 91.043,A -85,B 0,C 180,E1 -15619.874,E2 -15619.874} C_VEL
LIN {X 0,Y 312.537,Z 91.048,A -85,B 0,C 180,E1 -15624.05,E2 -15624.05} C_VEL
LIN {X 0,Y 312.505,Z 91.047,A -85,B 0,C 180,E1 -15627.333,E2 -15627.333} C_VEL
LIN {X 0,Y 312.545,Z 91.04,A -85,B 0,C 180,E1 -15631.278,E2 -15631.278} C_VEL
LIN {X 0,Y 312.587,Z 91.032,A -85,B 0,C 180,E1 -15634.71,E2 -15634.71} C_VEL
LIN {X 0,Y 312.588,Z 91.043,A -85,B 0,C 180,E1 -15637.528,E2 -15637.528} C_VEL
LIN {X 0,Y 312.639,Z 91.008,A -85,B 0,C 180,E1 -15641.656,E2 -15641.656} C_VEL
LIN {X 0,Y 312.694,Z 91.031,A -85,B 0,C 180,E1 -15645.686,E2 -15645.686} C_VEL
LIN {X 0,Y 312.702,Z 91,A -85,B 0,C 180,E1 -15649.641,E2 -15649.641} C_VEL
LIN {X 0,Y 312.873,Z 90.992,A -85,B 0,C 180,E1 -15652.254,E2 -15652.254} C_VEL
LIN {X 0,Y 312.719,Z 91.03,A -85,B 0,C 180,E1 -15654.842,E2 -15654.842} C_VEL
LIN {X 0,Y 312.988,Z 90.972,A -85,B 0,C 180,E1 -15658.713,E2 -15658.713} C_VEL
LIN {X 0,Y 312.988,Z 90.97,A -85,B 0,C 180,E1 -15661.286,E2 -15661.286} C_VEL
LIN {X 0,Y 312.717,Z 91.031,A -85,B 0,C 180,E1 -15665.157,E2 -15665.157} C_VEL
LIN {X 0,Y 312.871,Z 90.994,A -85,B 0,C 180,E1 -15667.745,E2 -15667.745} C_VEL
LIN {X 0,Y 312.671,Z 91.017,A -85,B 0,C 180,E1 -15671.67,E2 -15671.67} C_VEL
LIN {X 0,Y 312.699,Z 91.033,A -85,B 0,C 180,E1 -15674.887,E2 -15674.887} C_VEL
LIN {X 0,Y 312.628,Z 91.012,A -85,B 0,C 180,E1 -15679.236,E2 -15679.236} C_VEL
LIN {X 0,Y 312.544,Z 91.052,A -85,B 0,C 180,E1 -15682.789,E2 -15682.789} C_VEL
LIN {X 0,Y 312.6,Z 91.031,A -85,B 0,C 180,E1 -15685.935,E2 -15685.935} C_VEL
LIN {X 0,Y 312.535,Z 91.051,A -85,B 0,C 180,E1 -15689.65,E2 -15689.65} C_VEL
LIN {X 0,Y 312.517,Z 91.04,A -85,B 0,C 180,E1 -15693.688,E2 -15693.688} C_VEL
LIN {X 0,Y 312.538,Z 91.055,A -85,B 0,C 180,E1 -15697.382,E2 -15697.382} C_VEL
LIN {X 0,Y 312.497,Z 91.044,A -85,B 0,C 180,E1 -15700.707,E2 -15700.707} C_VEL
LIN {X 0,Y 312.452,Z 91.062,A -85,B 0,C 180,E1 -15704.208,E2 -15704.208} C_VEL
LIN {X 0,Y 312.48,Z 91.01,A -85,B 0,C 180,E1 -15707.918,E2 -15707.918} C_VEL
LIN {X 0,Y 312.531,Z 91.057,A -85,B 0,C 180,E1 -15711.91,E2 -15711.91} C_VEL
LIN {X 0,Y 312.502,Z 91.026,A -85,B 0,C 180,E1 -15715.79,E2 -15715.79} C_VEL
LIN {X 0,Y 312.517,Z 91.053,A -85,B 0,C 180,E1 -15718.853,E2 -15718.853} C_VEL
LIN {X 0,Y 312.566,Z 91.035,A -85,B 0,C 180,E1 -15721.824,E2 -15721.824} C_VEL
LIN {X 0,Y 312.603,Z 91.216,A -85,B 0,C 180,E1 -15723.741,E2 -15723.741} C_VEL
LIN {X 0,Y 312.824,Z 92.095,A -85,B 0,C 180,E1 -15723.98,E2 -15723.98} C_VEL
LIN {X 0,Y 314.288,Z 94.863,A -85,B 0,C 180,E1 -15724.26,E2 -15724.26} C_VEL
LIN {X 0,Y 317.383,Z 99.444,A -85,B 0,C 180,E1 -15724.753,E2 -15724.753} C_VEL
LIN {X 0,Y 320.651,Z 104.136,A -85,B 0,C 180,E1 -15725.323,E2 -15725.323} C_VEL
LIN {X 0,Y 325.311,Z 109.812,A -85,B 0,C 180,E1 -15726.15,E2 -15726.15} C_VEL
LIN {X 0,Y 330.102,Z 115.429,A -85,B 0,C 180,E1 -15727.068,E2 -15727.068} C_VEL
LIN {X 0,Y 335.059,Z 121.052,A -85,B 0,C 180,E1 -15728.075,E2 -15728.075} C_VEL
LIN {X 0,Y 341.132,Z 127.405,A -85,B 0,C 180,E1 -15729.382,E2 -15729.382} C_VEL
LIN {X 0,Y 347.249,Z 133.613,A -85,B 0,C 180,E1 -15730.798,E2 -15730.798} C_VEL
LIN {X 0,Y 350.481,Z 136.708,A -85,B 0,C 180,E1 -15731.604,E2 -15731.604} C_VEL
LIN {X 0,Y 355.261,Z 140.951,A -85,B 0,C 180,E1 -15732.838,E2 -15732.838} C_VEL
LIN {X 0,Y 357.772,Z 143.168,A -85,B 0,C 180,E1 -15733.525,E2 -15733.525} C_VEL
LIN {X 0,Y 362.396,Z 147.38,A -85,B 0,C 180,E1 -15734.895,E2 -15734.895} C_VEL
LIN {X 0,Y 366.013,Z 150.226,A -85,B 0,C 180,E1 -15736.053,E2 -15736.053} C_VEL
LIN {X 0,Y 370.19,Z 154.021,A -85,B 0,C 180,E1 -15737.548,E2 -15737.548} C_VEL
LIN {X 0,Y 373.945,Z 156.547,A -85,B 0,C 180,E1 -15739.03,E2 -15739.03} C_VEL
LIN {X 0,Y 375.882,Z 157.798,A -85,B 0,C 180,E1 -15739.873,E2 -15739.873} C_VEL
LIN {X 0,Y 378.948,Z 160.873,A -85,B 0,C 180,E1 -15741.468,E2 -15741.468} C_VEL
LIN {X 0,Y 381.669,Z 162.907,A -85,B 0,C 180,E1 -15743.143,E2 -15743.143} C_VEL
LIN {X 0,Y 384.063,Z 164.236,A -85,B 0,C 180,E1 -15745.023,E2 -15745.023} C_VEL
LIN {X 0,Y 385.734,Z 164.806,A -85,B 0,C 180,E1 -15746.867,E2 -15746.867} C_VEL
LIN {X 0,Y 386.667,Z 165.415,A -85,B 0,C 180,E1 -15748.959,E2 -15748.959} C_VEL
LIN {X 0,Y 386.811,Z 165.321,A -85,B 0,C 180,E1 -15750,E2 -15750} C_VEL
LIN {X 0,Y 386.523,Z 165.254,A -85,B 0,C 180,E1 -15751.563,E2 -15751.563} C_VEL
LIN {X 0,Y 385.729,Z 164.835,A -85,B 0,C 180,E1 -15753.133,E2 -15753.133} C_VEL
LIN {X 0,Y 384.063,Z 164.236,A -85,B 0,C 180,E1 -15754.977,E2 -15754.977} C_VEL
LIN {X 0,Y 381.669,Z 162.909,A -85,B 0,C 180,E1 -15756.856,E2 -15756.856} C_VEL
LIN {X 0,Y 378.692,Z 160.653,A -85,B 0,C 180,E1 -15758.683,E2 -15758.683} C_VEL
LIN {X 0,Y 375.155,Z 157.179,A -85,B 0,C 180,E1 -15760.465,E2 -15760.465} C_VEL
LIN {X 0,Y 371.149,Z 154.689,A -85,B 0,C 180,E1 -15762.097,E2 -15762.097} C_VEL
LIN {X 0,Y 367.011,Z 151.186,A -85,B 0,C 180,E1 -15763.611,E2 -15763.611} C_VEL
LIN {X 0,Y 363.841,Z 148.441,A -85,B 0,C 180,E1 -15764.661,E2 -15764.661} C_VEL
LIN {X 0,Y 358.945,Z 144.379,A -85,B 0,C 180,E1 -15766.135,E2 -15766.135} C_VEL
LIN {X 0,Y 355.764,Z 141.319,A -85,B 0,C 180,E1 -15767.026,E2 -15767.026} C_VEL
LIN {X 0,Y 351.292,Z 137.541,A -85,B 0,C 180,E1 -15768.191,E2 -15768.191} C_VEL
LIN {X 0,Y 347.696,Z 133.958,A -85,B 0,C 180,E1 -15769.095,E2 -15769.095} C_VEL
LIN {X 0,Y 343.066,Z 129.451,A -85,B 0,C 180,E1 -15770.174,E2 -15770.174} C_VEL
LIN {X 0,Y 336.603,Z 122.689,A -85,B 0,C 180,E1 -15771.594,E2 -15771.594} C_VEL
LIN {X 0,Y 331.27,Z 116.884,A -85,B 0,C 180,E1 -15772.69,E2 -15772.69} C_VEL
LIN {X 0,Y 326.098,Z 110.761,A -85,B 0,C 180,E1 -15773.701,E2 -15773.701} C_VEL
LIN {X 0,Y 322.079,Z 105.836,A -85,B 0,C 180,E1 -15774.438,E2 -15774.438} C_VEL
LIN {X 0,Y 318.2,Z 100.775,A -85,B 0,C 180,E1 -15775.104,E2 -15775.104} C_VEL
LIN {X 0,Y 314.856,Z 95.626,A -85,B 0,C 180,E1 -15775.652,E2 -15775.652} C_VEL
LIN {X 0,Y 313.013,Z 92.734,A -85,B 0,C 180,E1 -15775.959,E2 -15775.959} C_VEL
LIN {X 0,Y 312.643,Z 91.414,A -85,B 0,C 180,E1 -15776.16,E2 -15776.16} C_VEL
LIN {X 0,Y 312.549,Z 91.054,A -85,B 0,C 180,E1 -15776.726,E2 -15776.726} C_VEL
LIN {X 0,Y 312.534,Z 91.032,A -85,B 0,C 180,E1 -15779.651,E2 -15779.651} C_VEL
LIN {X 0,Y 312.516,Z 91.027,A -85,B 0,C 180,E1 -15783.689,E2 -15783.689} C_VEL
LIN {X 0,Y 312.534,Z 91.053,A -85,B 0,C 180,E1 -15787.384,E2 -15787.384} C_VEL
LIN {X 0,Y 312.486,Z 91.02,A -85,B 0,C 180,E1 -15790.71,E2 -15790.71} C_VEL
LIN {X 0,Y 312.449,Z 91.038,A -85,B 0,C 180,E1 -15794.21,E2 -15794.21} C_VEL
LIN {X 0,Y 312.522,Z 91.049,A -85,B 0,C 180,E1 -15797.911,E2 -15797.911} C_VEL
LIN {X 0,Y 312.54,Z 91.055,A -85,B 0,C 180,E1 -15801.909,E2 -15801.909} C_VEL
LIN {X 0,Y 312.503,Z 91.039,A -85,B 0,C 180,E1 -15805.791,E2 -15805.791} C_VEL
LIN {X 0,Y 312.518,Z 91.058,A -85,B 0,C 180,E1 -15808.854,E2 -15808.854} C_VEL
LIN {X 0,Y 312.567,Z 91.03,A -85,B 0,C 180,E1 -15811.825,E2 -15811.825} C_VEL
LIN {X 0,Y 312.583,Z 91.037,A -85,B 0,C 180,E1 -15814.712,E2 -15814.712} C_VEL
LIN {X 0,Y 312.586,Z 91.045,A -85,B 0,C 180,E1 -15817.53,E2 -15817.53} C_VEL
LIN {X 0,Y 312.637,Z 91.013,A -85,B 0,C 180,E1 -15821.657,E2 -15821.657} C_VEL
LIN {X 0,Y 312.693,Z 91.033,A -85,B 0,C 180,E1 -15825.687,E2 -15825.687} C_VEL
LIN {X 0,Y 312.702,Z 91,A -85,B 0,C 180,E1 -15829.643,E2 -15829.643} C_VEL
LIN {X 0,Y 312.871,Z 90.994,A -85,B 0,C 180,E1 -15832.255,E2 -15832.255} C_VEL
LIN {X 0,Y 312.717,Z 91.031,A -85,B 0,C 180,E1 -15834.843,E2 -15834.843} C_VEL
LIN {X 0,Y 312.718,Z 91.026,A -85,B 0,C 180,E1 -15836.325,E2 -15836.325} C_VEL
LIN {X 0,Y 312.188,Z 91.086,A -85,B 0,C 180,E1 -15837.403,E2 -15837.403} C_VEL
LIN {X 0,Y 309.455,Z 91.408,A -85,B 0,C 180,E1 -15839.161,E2 -15839.161} C_VEL
LIN {X 0,Y 307.051,Z 91.706,A -85,B 0,C 180,E1 -15840.586,E2 -15840.586} C_VEL
LIN {X 0,Y 305.992,Z 91.846,A -85,B 0,C 180,E1 -15841.688,E2 -15841.688} C_VEL
LIN {X 0,Y 305.896,Z 91.862,A -85,B 0,C 180,E1 -15842.062,E2 -15842.062} C_VEL
LIN {X 0,Y 305.854,Z 91.879,A -85,B 0,C 180,E1 -15846.598,E2 -15846.598} C_VEL
LIN {X 0,Y 305.736,Z 91.865,A -85,B 0,C 180,E1 -15849.26,E2 -15849.26} C_VEL
LIN {X 0,Y 305.59,Z 91.913,A -85,B 0,C 180,E1 -15853.297,E2 -15853.297} C_VEL
LIN {X 0,Y 305.594,Z 91.908,A -85,B 0,C 180,E1 -15856.021,E2 -15856.021} C_VEL
LIN {X 0,Y 305.577,Z 91.888,A -85,B 0,C 180,E1 -15859.445,E2 -15859.445} C_VEL
LIN {X 0,Y 305.492,Z 91.93,A -85,B 0,C 180,E1 -15863.042,E2 -15863.042} C_VEL
LIN {X 0,Y 305.532,Z 91.903,A -85,B 0,C 180,E1 -15866.221,E2 -15866.221} C_VEL
LIN {X 0,Y 305.489,Z 91.921,A -85,B 0,C 180,E1 -15869.048,E2 -15869.048} C_VEL
LIN {X 0,Y 305.444,Z 91.934,A -85,B 0,C 180,E1 -15871.953,E2 -15871.953} C_VEL
LIN {X 0,Y 305.464,Z 91.917,A -85,B 0,C 180,E1 -15875.114,E2 -15875.114} C_VEL
LIN {X 0,Y 305.451,Z 91.933,A -85,B 0,C 180,E1 -15878.529,E2 -15878.529} C_VEL
LIN {X 0,Y 305.457,Z 91.939,A -85,B 0,C 180,E1 -15882.586,E2 -15882.586} C_VEL
LIN {X 0,Y 305.427,Z 91.939,A -85,B 0,C 180,E1 -15886.345,E2 -15886.345} C_VEL
LIN {X 0,Y 305.46,Z 91.905,A -85,B 0,C 180,E1 -15889.893,E2 -15889.893} C_VEL
LIN {X 0,Y 305.502,Z 91.918,A -85,B 0,C 180,E1 -15893.627,E2 -15893.627} C_VEL
LIN {X 0,Y 305.524,Z 92.152,A -85,B 0,C 180,E1 -15895.193,E2 -15895.193} C_VEL
LIN {X 0,Y 307.075,Z 99.502,A -85,B 0,C 180,E1 -15898.238,E2 -15898.238} C_VEL
LIN {X 0,Y 308.917,Z 109,A -85,B 0,C 180,E1 -15902.057,E2 -15902.057} C_VEL
LIN {X 0,Y 309.065,Z 113.309,A -85,B 0,C 180,E1 -15903.64,E2 -15903.64} C_VEL
LIN {X 0,Y 309.745,Z 116.887,A -85,B 0,C 180,E1 -15903.869,E2 -15903.869} C_VEL
LIN {X 0,Y 314.835,Z 140.612,A -85,B 0,C 180,E1 -15904.904,E2 -15904.904} C_VEL
LIN {X 0,Y 317.566,Z 156.538,A -85,B 0,C 180,E1 -15905.521,E2 -15905.521} C_VEL
LIN {X 0,Y 316.157,Z 218.207,A -85,B 0,C 180,E1 -15906.934,E2 -15906.934} C_VEL
LIN {X 0,Y 315.542,Z 228.918,A -85,B 0,C 180,E1 -15907.319,E2 -15907.319} C_VEL
LIN {X 0,Y 314.761,Z 238.017,A -85,B 0,C 180,E1 -15907.779,E2 -15907.779} C_VEL
LIN {X 0,Y 313.752,Z 248.378,A -85,B 0,C 180,E1 -15908.482,E2 -15908.482} C_VEL
LIN {X 0,Y 312.658,Z 257.509,A -85,B 0,C 180,E1 -15909.266,E2 -15909.266} C_VEL
LIN {X 0,Y 311.436,Z 266.503,A -85,B 0,C 180,E1 -15910.215,E2 -15910.215} C_VEL
LIN {X 0,Y 310.176,Z 275.23,A -85,B 0,C 180,E1 -15911.334,E2 -15911.334} C_VEL
LIN {X 0,Y 309.019,Z 282.623,A -85,B 0,C 180,E1 -15912.462,E2 -15912.462} C_VEL
LIN {X 0,Y 307.967,Z 289.932,A -85,B 0,C 180,E1 -15913.785,E2 -15913.785} C_VEL
LIN {X 0,Y 307.022,Z 296.047,A -85,B 0,C 180,E1 -15915.077,E2 -15915.077} C_VEL
LIN {X 0,Y 305.936,Z 302.583,A -85,B 0,C 180,E1 -15916.719,E2 -15916.719} C_VEL
LIN {X 0,Y 305.18,Z 307.083,A -85,B 0,C 180,E1 -15918.038,E2 -15918.038} C_VEL
LIN {X 0,Y 304.45,Z 312.576,A -85,B 0,C 180,E1 -15920.03,E2 -15920.03} C_VEL
LIN {X 0,Y 303.958,Z 316.903,A -85,B 0,C 180,E1 -15922.026,E2 -15922.026} C_VEL
LIN {X 0,Y 303.743,Z 319.271,A -85,B 0,C 180,E1 -15923.357,E2 -15923.357} C_VEL
LIN {X 0,Y 303.62,Z 321.071,A -85,B 0,C 180,E1 -15924.687,E2 -15924.687} C_VEL
LIN {X 0,Y 303.603,Z 323.521,A -85,B 0,C 180,E1 -15927.346,E2 -15927.346} C_VEL
LIN {X 0,Y 303.566,Z 324.11,A -85,B 0,C 180,E1 -15928.673,E2 -15928.673} C_VEL
LIN {X 0,Y 303.566,Z 324.11,A -85,B 0,C 180,E1 -15931.327,E2 -15931.327} C_VEL
LIN {X 0,Y 303.603,Z 323.521,A -85,B 0,C 180,E1 -15932.654,E2 -15932.654} C_VEL
LIN {X 0,Y 303.62,Z 321.071,A -85,B 0,C 180,E1 -15935.313,E2 -15935.313} C_VEL
LIN {X 0,Y 303.841,Z 318.12,A -85,B 0,C 180,E1 -15937.309,E2 -15937.309} C_VEL
LIN {X 0,Y 304.265,Z 314.131,A -85,B 0,C 180,E1 -15939.305,E2 -15939.305} C_VEL
LIN {X 0,Y 304.915,Z 308.999,A -85,B 0,C 180,E1 -15941.298,E2 -15941.298} C_VEL
LIN {X 0,Y 305.724,Z 303.737,A -85,B 0,C 180,E1 -15942.952,E2 -15942.952} C_VEL
LIN {X 0,Y 306.783,Z 297.422,A -85,B 0,C 180,E1 -15944.596,E2 -15944.596} C_VEL
LIN {X 0,Y 307.75,Z 291.472,A -85,B 0,C 180,E1 -15945.905,E2 -15945.905} C_VEL
LIN {X 0,Y 308.76,Z 284.543,A -85,B 0,C 180,E1 -15947.212,E2 -15947.212} C_VEL
LIN {X 0,Y 310.003,Z 276.364,A -85,B 0,C 180,E1 -15948.505,E2 -15948.505} C_VEL
LIN {X 0,Y 311.26,Z 267.855,A -85,B 0,C 180,E1 -15949.625,E2 -15949.625} C_VEL
LIN {X 0,Y 312.459,Z 259.141,A -85,B 0,C 180,E1 -15950.576,E2 -15950.576} C_VEL
LIN {X 0,Y 313.631,Z 249.385,A -85,B 0,C 180,E1 -15951.441,E2 -15951.441} C_VEL
LIN {X 0,Y 314.67,Z 239.305,A -85,B 0,C 180,E1 -15952.141,E2 -15952.141} C_VEL
LIN {X 0,Y 315.484,Z 229.792,A -85,B 0,C 180,E1 -15952.642,E2 -15952.642} C_VEL
LIN {X 0,Y 316.024,Z 219.478,A -85,B 0,C 180,E1 -15953.033,E2 -15953.033} C_VEL
LIN {X 0,Y 317.059,Z 178.797,A -85,B 0,C 180,E1 -15953.98,E2 -15953.98} C_VEL
LIN {X 0,Y 317.477,Z 155.838,A -85,B 0,C 180,E1 -15954.504,E2 -15954.504} C_VEL
LIN {X 0,Y 312.93,Z 131.049,A -85,B 0,C 180,E1 -15955.495,E2 -15955.495} C_VEL
LIN {X 0,Y 309.066,Z 113.668,A -85,B 0,C 180,E1 -15956.308,E2 -15956.308} C_VEL
LIN {X 0,Y 309.122,Z 112.249,A -85,B 0,C 180,E1 -15956.681,E2 -15956.681} C_VEL
LIN {X 0,Y 308.622,Z 107.436,A -85,B 0,C 180,E1 -15958.569,E2 -15958.569} C_VEL
LIN {X 0,Y 306.675,Z 97.33,A -85,B 0,C 180,E1 -15962.643,E2 -15962.643} C_VEL
LIN {X 0,Y 305.519,Z 91.945,A -85,B 0,C 180,E1 -15964.97,E2 -15964.97} C_VEL
LIN {X 0,Y 305.469,Z 91.919,A -85,B 0,C 180,E1 -15968.532,E2 -15968.532} C_VEL
LIN {X 0,Y 305.457,Z 91.935,A -85,B 0,C 180,E1 -15972.585,E2 -15972.585} C_VEL
LIN {X 0,Y 305.427,Z 91.938,A -85,B 0,C 180,E1 -15976.344,E2 -15976.344} C_VEL
LIN {X 0,Y 305.46,Z 91.921,A -85,B 0,C 180,E1 -15979.892,E2 -15979.892} C_VEL
LIN {X 0,Y 305.483,Z 91.928,A -85,B 0,C 180,E1 -15983.631,E2 -15983.631} C_VEL
LIN {X 0,Y 305.466,Z 91.915,A -85,B 0,C 180,E1 -15986.483,E2 -15986.483} C_VEL
LIN {X 0,Y 305.459,Z 91.934,A -85,B 0,C 180,E1 -15989.59,E2 -15989.59} C_VEL
LIN {X 0,Y 305.519,Z 91.902,A -85,B 0,C 180,E1 -15992.608,E2 -15992.608} C_VEL
LIN {X 0,Y 305.509,Z 91.924,A -85,B 0,C 180,E1 -15995.538,E2 -15995.538} C_VEL
LIN {X 0,Y 305.52,Z 91.904,A -85,B 0,C 180,E1 -15999.814,E2 -15999.814} C_VEL
LIN {X 0,Y 305.575,Z 91.895,A -85,B 0,C 180,E1 -16002.602,E2 -16002.602} C_VEL
LIN {X 0,Y 305.65,Z 91.908,A -85,B 0,C 180,E1 -16005.348,E2 -16005.348} C_VEL
LIN {X 0,Y 305.639,Z 91.881,A -85,B 0,C 180,E1 -16009.399,E2 -16009.399} C_VEL
LIN {X 0,Y 305.814,Z 91.868,A -85,B 0,C 180,E1 -16012.074,E2 -16012.074} C_VEL
LIN {X 0,Y 305.69,Z 91.906,A -85,B 0,C 180,E1 -16014.723,E2 -16014.723} C_VEL
LIN {X 0,Y 305.955,Z 91.848,A -85,B 0,C 180,E1 -16018.683,E2 -16018.683} C_VEL
LIN {X 0,Y 305.955,Z 91.845,A -85,B 0,C 180,E1 -16021.316,E2 -16021.316} C_VEL
LIN {X 0,Y 305.851,Z 91.88,A -85,B 0,C 180,E1 -16026.605,E2 -16026.605} C_VEL
LIN {X 0,Y 305.735,Z 91.867,A -85,B 0,C 180,E1 -16029.259,E2 -16029.259} C_VEL
LIN {X 0,Y 305.59,Z 91.915,A -85,B 0,C 180,E1 -16033.295,E2 -16033.295} C_VEL
LIN {X 0,Y 305.592,Z 91.913,A -85,B 0,C 180,E1 -16036.019,E2 -16036.019} C_VEL
LIN {X 0,Y 305.575,Z 91.89,A -85,B 0,C 180,E1 -16039.444,E2 -16039.444} C_VEL
LIN {X 0,Y 305.489,Z 91.932,A -85,B 0,C 180,E1 -16043.041,E2 -16043.041} C_VEL
LIN {X 0,Y 305.529,Z 91.907,A -85,B 0,C 180,E1 -16046.22,E2 -16046.22} C_VEL
LIN {X 0,Y 305.485,Z 91.92,A -85,B 0,C 180,E1 -16049.047,E2 -16049.047} C_VEL
LIN {X 0,Y 305.44,Z 91.937,A -85,B 0,C 180,E1 -16051.952,E2 -16051.952} C_VEL
LIN {X 0,Y 305.46,Z 91.918,A -85,B 0,C 180,E1 -16055.113,E2 -16055.113} C_VEL
LIN {X 0,Y 305.48,Z 91.932,A -85,B 0,C 180,E1 -16058.536,E2 -16058.536} C_VEL
LIN {X 0,Y 305.48,Z 91.931,A -85,B 0,C 180,E1 -16062.591,E2 -16062.591} C_VEL
LIN {X 0,Y 305.451,Z 91.886,A -85,B 0,C 180,E1 -16067.414,E2 -16067.414} C_VEL
LIN {X 0,Y 305.491,Z 91.932,A -85,B 0,C 180,E1 -16071.6,E2 -16071.6} C_VEL
LIN {X 0,Y 305.459,Z 91.902,A -85,B 0,C 180,E1 -16074.886,E2 -16074.886} C_VEL
LIN {X 0,Y 305.446,Z 91.939,A -85,B 0,C 180,E1 -16078.355,E2 -16078.355} C_VEL
LIN {X 0,Y 305.509,Z 91.907,A -85,B 0,C 180,E1 -16081.113,E2 -16081.113} C_VEL
LIN {X 0,Y 305.528,Z 92.083,A -85,B 0,C 180,E1 -16082.989,E2 -16082.989} C_VEL
LIN {X 0,Y 305.764,Z 93.092,A -85,B 0,C 180,E1 -16083.25,E2 -16083.25} C_VEL
LIN {X 0,Y 309.458,Z 99.513,A -85,B 0,C 180,E1 -16083.829,E2 -16083.829} C_VEL
LIN {X 0,Y 315.161,Z 107.845,A -85,B 0,C 180,E1 -16084.712,E2 -16084.712} C_VEL
LIN {X 0,Y 321.519,Z 115.383,A -85,B 0,C 180,E1 -16085.752,E2 -16085.752} C_VEL
LIN {X 0,Y 326.493,Z 121.071,A -85,B 0,C 180,E1 -16086.657,E2 -16086.657} C_VEL
LIN {X 0,Y 331.627,Z 126.789,A -85,B 0,C 180,E1 -16087.661,E2 -16087.661} C_VEL
LIN {X 0,Y 337.794,Z 133.178,A -85,B 0,C 180,E1 -16088.948,E2 -16088.948} C_VEL
LIN {X 0,Y 344.045,Z 139.408,A -85,B 0,C 180,E1 -16090.343,E2 -16090.343} C_VEL
LIN {X 0,Y 347.95,Z 142.982,A -85,B 0,C 180,E1 -16091.26,E2 -16091.26} C_VEL
LIN {X 0,Y 352.951,Z 147.364,A -85,B 0,C 180,E1 -16092.517,E2 -16092.517} C_VEL
LIN {X 0,Y 356.987,Z 151.039,A -85,B 0,C 180,E1 -16093.617,E2 -16093.617} C_VEL
LIN {X 0,Y 361.827,Z 155.008,A -85,B 0,C 180,E1 -16095.039,E2 -16095.039} C_VEL
LIN {X 0,Y 364.855,Z 157.511,A -85,B 0,C 180,E1 -16096.008,E2 -16096.008} C_VEL
LIN {X 0,Y 368.937,Z 161.021,A -85,B 0,C 180,E1 -16097.445,E2 -16097.445} C_VEL
LIN {X 0,Y 372.723,Z 163.498,A -85,B 0,C 180,E1 -16098.914,E2 -16098.914} C_VEL
LIN {X 0,Y 374.583,Z 164.71,A -85,B 0,C 180,E1 -16099.701,E2 -16099.701} C_VEL
LIN {X 0,Y 377.883,Z 167.882,A -85,B 0,C 180,E1 -16101.376,E2 -16101.376} C_VEL
LIN {X 0,Y 380.706,Z 169.936,A -85,B 0,C 180,E1 -16103.09,E2 -16103.09} C_VEL
LIN {X 0,Y 383.173,Z 171.282,A -85,B 0,C 180,E1 -16105.011,E2 -16105.011} C_VEL
LIN {X 0,Y 384.859,Z 171.829,A -85,B 0,C 180,E1 -16106.86,E2 -16106.86} C_VEL
LIN {X 0,Y 385.802,Z 172.461,A -85,B 0,C 180,E1 -16108.956,E2 -16108.956} C_VEL
LIN {X 0,Y 385.946,Z 172.368,A -85,B 0,C 180,E1 -16110,E2 -16110} C_VEL
LIN {X 0,Y 385.654,Z 172.302,A -85,B 0,C 180,E1 -16111.566,E2 -16111.566} C_VEL
LIN {X 0,Y 384.853,Z 171.87,A -85,B 0,C 180,E1 -16113.14,E2 -16113.14} C_VEL
LIN {X 0,Y 383.173,Z 171.281,A -85,B 0,C 180,E1 -16114.989,E2 -16114.989} C_VEL
LIN {X 0,Y 380.706,Z 169.938,A -85,B 0,C 180,E1 -16116.91,E2 -16116.91} C_VEL
LIN {X 0,Y 377.565,Z 167.644,A -85,B 0,C 180,E1 -16118.792,E2 -16118.792} C_VEL
LIN {X 0,Y 373.598,Z 163.955,A -85,B 0,C 180,E1 -16120.732,E2 -16120.732} C_VEL
LIN {X 0,Y 369.7,Z 161.565,A -85,B 0,C 180,E1 -16122.277,E2 -16122.277} C_VEL
LIN {X 0,Y 365.262,Z 157.899,A -85,B 0,C 180,E1 -16123.856,E2 -16123.856} C_VEL
LIN {X 0,Y 362.05,Z 155.151,A -85,B 0,C 180,E1 -16124.893,E2 -16124.893} C_VEL
LIN {X 0,Y 356.986,Z 151.061,A -85,B 0,C 180,E1 -16126.382,E2 -16126.382} C_VEL
LIN {X 0,Y 353.196,Z 147.517,A -85,B 0,C 180,E1 -16127.421,E2 -16127.421} C_VEL
LIN {X 0,Y 348.374,Z 143.426,A -85,B 0,C 180,E1 -16128.636,E2 -16128.636} C_VEL
LIN {X 0,Y 345.059,Z 140.252,A -85,B 0,C 180,E1 -16129.429,E2 -16129.429} C_VEL
LIN {X 0,Y 340.07,Z 135.446,A -85,B 0,C 180,E1 -16130.568,E2 -16130.568} C_VEL
LIN {X 0,Y 333.452,Z 128.672,A -85,B 0,C 180,E1 -16131.974,E2 -16131.974} C_VEL
LIN {X 0,Y 327.605,Z 122.421,A -85,B 0,C 180,E1 -16133.128,E2 -16133.128} C_VEL
LIN {X 0,Y 321.997,Z 115.925,A -85,B 0,C 180,E1 -16134.165,E2 -16134.165} C_VEL
LIN {X 0,Y 317.523,Z 110.565,A -85,B 0,C 180,E1 -16134.919,E2 -16134.919} C_VEL
LIN {X 0,Y 313.703,Z 105.782,A -85,B 0,C 180,E1 -16135.517,E2 -16135.517} C_VEL
LIN {X 0,Y 308.301,Z 97.826,A -85,B 0,C 180,E1 -16136.334,E2 -16136.334} C_VEL
LIN {X 0,Y 305.762,Z 93.099,A -85,B 0,C 180,E1 -16136.749,E2 -16136.749} C_VEL
LIN {X 0,Y 305.528,Z 92.085,A -85,B 0,C 180,E1 -16137.01,E2 -16137.01} C_VEL
LIN {X 0,Y 305.454,Z 91.92,A -85,B 0,C 180,E1 -16140.41,E2 -16140.41} C_VEL
LIN {X 0,Y 305.461,Z 91.902,A -85,B 0,C 180,E1 -16144.079,E2 -16144.079} C_VEL
LIN {X 0,Y 305.492,Z 91.92,A -85,B 0,C 180,E1 -16146.737,E2 -16146.737} C_VEL
LIN {X 0,Y 305.451,Z 91.897,A -85,B 0,C 180,E1 -16150.6,E2 -16150.6} C_VEL
LIN {X 0,Y 305.422,Z 91.902,A -85,B 0,C 180,E1 -16153.656,E2 -16153.656} C_VEL
LIN {X 0,Y 305.48,Z 91.931,A -85,B 0,C 180,E1 -16157.409,E2 -16157.409} C_VEL
LIN {X 0,Y 305.506,Z 91.931,A -85,B 0,C 180,E1 -16161.603,E2 -16161.603} C_VEL
LIN {X 0,Y 305.46,Z 91.918,A -85,B 0,C 180,E1 -16164.887,E2 -16164.887} C_VEL
LIN {X 0,Y 305.447,Z 91.936,A -85,B 0,C 180,E1 -16168.356,E2 -16168.356} C_VEL
LIN {X 0,Y 305.51,Z 91.915,A -85,B 0,C 180,E1 -16171.114,E2 -16171.114} C_VEL
LIN {X 0,Y 305.569,Z 91.906,A -85,B 0,C 180,E1 -16174.089,E2 -16174.089} C_VEL
LIN {X 0,Y 305.498,Z 91.923,A -85,B 0,C 180,E1 -16178.404,E2 -16178.404} C_VEL
LIN {X 0,Y 305.588,Z 91.888,A -85,B 0,C 180,E1 -16181.218,E2 -16181.218} C_VEL
LIN {X 0,Y 305.648,Z 91.911,A -85,B 0,C 180,E1 -16185.35,E2 -16185.35} C_VEL
LIN {X 0,Y 305.639,Z 91.881,A -85,B 0,C 180,E1 -16189.401,E2 -16189.401} C_VEL
LIN {X 0,Y 305.812,Z 91.871,A -85,B 0,C 180,E1 -16192.075,E2 -16192.075} C_VEL
LIN {X 0,Y 305.688,Z 91.907,A -85,B 0,C 180,E1 -16194.724,E2 -16194.724} C_VEL
LIN {X 0,Y 305.955,Z 91.845,A -85,B 0,C 180,E1 -16198.684,E2 -16198.684} C_VEL
LIN {X 0,Y 305.955,Z 91.848,A -85,B 0,C 180,E1 -16201.317,E2 -16201.317} C_VEL
LIN {X 0,Y 305.896,Z 91.862,A -85,B 0,C 180,E1 -16202.062,E2 -16202.062} C_VEL
LIN {X 0,Y 305.191,Z 91.963,A -85,B 0,C 180,E1 -16203.159,E2 -16203.159} C_VEL
LIN {X 0,Y 302.293,Z 92.329,A -85,B 0,C 180,E1 -16204.944,E2 -16204.944} C_VEL
LIN {X 0,Y 299.861,Z 92.626,A -85,B 0,C 180,E1 -16206.392,E2 -16206.392} C_VEL
LIN {X 0,Y 298.832,Z 92.742,A -85,B 0,C 180,E1 -16207.515,E2 -16207.515} C_VEL
LIN {X 0,Y 298.755,Z 92.747,A -85,B 0,C 180,E1 -16207.895,E2 -16207.895} C_VEL
LIN {X 0,Y 298.594,Z 92.76,A -85,B 0,C 180,E1 -16210.854,E2 -16210.854} C_VEL
LIN {X 0,Y 298.606,Z 92.787,A -85,B 0,C 180,E1 -16215.21,E2 -16215.21} C_VEL
LIN {X 0,Y 298.54,Z 92.762,A -85,B 0,C 180,E1 -16219.244,E2 -16219.244} C_VEL
LIN {X 0,Y 298.459,Z 92.805,A -85,B 0,C 180,E1 -16223.598,E2 -16223.598} C_VEL
LIN {X 0,Y 298.488,Z 92.777,A -85,B 0,C 180,E1 -16226.575,E2 -16226.575} C_VEL
LIN {X 0,Y 298.418,Z 92.81,A -85,B 0,C 180,E1 -16229.642,E2 -16229.642} C_VEL
LIN {X 0,Y 298.396,Z 92.802,A -85,B 0,C 180,E1 -16232.801,E2 -16232.801} C_VEL
LIN {X 0,Y 298.448,Z 92.808,A -85,B 0,C 180,E1 -16236.808,E2 -16236.808} C_VEL
LIN {X 0,Y 298.389,Z 92.806,A -85,B 0,C 180,E1 -16241.088,E2 -16241.088} C_VEL
LIN {X 0,Y 298.401,Z 92.814,A -85,B 0,C 180,E1 -16243.104,E2 -16243.104} C_VEL
LIN {X 0,Y 298.405,Z 92.815,A -85,B 0,C 180,E1 -16246.921,E2 -16246.921} C_VEL
LIN {X 0,Y 298.417,Z 92.789,A -85,B 0,C 180,E1 -16251.004,E2 -16251.004} C_VEL
LIN {X 0,Y 298.502,Z 92.956,A -85,B 0,C 180,E1 -16254.655,E2 -16254.655} C_VEL
LIN {X 0,Y 300.238,Z 101.456,A -85,B 0,C 180,E1 -16258.29,E2 -16258.29} C_VEL
LIN {X 0,Y 301.738,Z 109.171,A -85,B 0,C 180,E1 -16261.48,E2 -16261.48} C_VEL
LIN {X 0,Y 302.198,Z 113.211,A -85,B 0,C 180,E1 -16263.014,E2 -16263.014} C_VEL
LIN {X 0,Y 303.506,Z 118.74,A -85,B 0,C 180,E1 -16263.342,E2 -16263.342} C_VEL
LIN {X 0,Y 308.495,Z 142.226,A -85,B 0,C 180,E1 -16264.397,E2 -16264.397} C_VEL
LIN {X 0,Y 311.097,Z 158.113,A -85,B 0,C 180,E1 -16265.021,E2 -16265.021} C_VEL
LIN {X 0,Y 309.58,Z 219.29,A -85,B 0,C 180,E1 -16266.459,E2 -16266.459} C_VEL
LIN {X 0,Y 308.949,Z 229.602,A -85,B 0,C 180,E1 -16266.852,E2 -16266.852} C_VEL
LIN {X 0,Y 308.1,Z 239.114,A -85,B 0,C 180,E1 -16267.361,E2 -16267.361} C_VEL
LIN {X 0,Y 307.048,Z 249.194,A -85,B 0,C 180,E1 -16268.076,E2 -16268.076} C_VEL
LIN {X 0,Y 305.804,Z 258.95,A -85,B 0,C 180,E1 -16268.955,E2 -16268.955} C_VEL
LIN {X 0,Y 304.358,Z 269.015,A -85,B 0,C 180,E1 -16270.087,E2 -16270.087} C_VEL
LIN {X 0,Y 302.533,Z 280.512,A -85,B 0,C 180,E1 -16271.723,E2 -16271.723} C_VEL
LIN {X 0,Y 301.261,Z 288.844,A -85,B 0,C 180,E1 -16273.221,E2 -16273.221} C_VEL
LIN {X 0,Y 300.107,Z 295.854,A -85,B 0,C 180,E1 -16274.725,E2 -16274.725} C_VEL
LIN {X 0,Y 299.003,Z 302.391,A -85,B 0,C 180,E1 -16276.406,E2 -16276.406} C_VEL
LIN {X 0,Y 298.207,Z 306.891,A -85,B 0,C 180,E1 -16277.754,E2 -16277.754} C_VEL
LIN {X 0,Y 297.43,Z 312.385,A -85,B 0,C 180,E1 -16279.792,E2 -16279.792} C_VEL
LIN {X 0,Y 296.898,Z 316.711,A -85,B 0,C 180,E1 -16281.835,E2 -16281.835} C_VEL
LIN {X 0,Y 296.69,Z 319.08,A -85,B 0,C 180,E1 -16283.198,E2 -16283.198} C_VEL
LIN {X 0,Y 296.534,Z 320.88,A -85,B 0,C 180,E1 -16284.56,E2 -16284.56} C_VEL
LIN {X 0,Y 296.528,Z 323.331,A -85,B 0,C 180,E1 -16287.283,E2 -16287.283} C_VEL
LIN {X 0,Y 296.486,Z 323.92,A -85,B 0,C 180,E1 -16288.642,E2 -16288.642} C_VEL
LIN {X 0,Y 296.486,Z 323.92,A -85,B 0,C 180,E1 -16291.358,E2 -16291.358} C_VEL
LIN {X 0,Y 296.528,Z 323.331,A -85,B 0,C 180,E1 -16292.717,E2 -16292.717} C_VEL
LIN {X 0,Y 296.549,Z 320.79,A -85,B 0,C 180,E1 -16295.509,E2 -16295.509} C_VEL
LIN {X 0,Y 296.79,Z 317.929,A -85,B 0,C 180,E1 -16297.483,E2 -16297.483} C_VEL
LIN {X 0,Y 297.237,Z 313.94,A -85,B 0,C 180,E1 -16299.527,E2 -16299.527} C_VEL
LIN {X 0,Y 297.915,Z 308.808,A -85,B 0,C 180,E1 -16301.567,E2 -16301.567} C_VEL
LIN {X 0,Y 298.793,Z 303.547,A -85,B 0,C 180,E1 -16303.258,E2 -16303.258} C_VEL
LIN {X 0,Y 299.872,Z 297.231,A -85,B 0,C 180,E1 -16304.94,E2 -16304.94} C_VEL
LIN {X 0,Y 300.917,Z 291.281,A -85,B 0,C 180,E1 -16306.276,E2 -16306.276} C_VEL
LIN {X 0,Y 301.967,Z 284.352,A -85,B 0,C 180,E1 -16307.612,E2 -16307.612} C_VEL
LIN {X 0,Y 303.272,Z 276.174,A -85,B 0,C 180,E1 -16308.931,E2 -16308.931} C_VEL
LIN {X 0,Y 304.554,Z 267.663,A -85,B 0,C 180,E1 -16310.076,E2 -16310.076} C_VEL
LIN {X 0,Y 305.819,Z 258.951,A -85,B 0,C 180,E1 -16311.043,E2 -16311.043} C_VEL
LIN {X 0,Y 307.018,Z 249.194,A -85,B 0,C 180,E1 -16311.926,E2 -16311.926} C_VEL
LIN {X 0,Y 307.994,Z 240.402,A -85,B 0,C 180,E1 -16312.559,E2 -16312.559} C_VEL
LIN {X 0,Y 308.89,Z 230.476,A -85,B 0,C 180,E1 -16313.109,E2 -16313.109} C_VEL
LIN {X 0,Y 309.452,Z 220.619,A -85,B 0,C 180,E1 -16313.507,E2 -16313.507} C_VEL
LIN {X 0,Y 310.151,Z 197.798,A -85,B 0,C 180,E1 -16314.072,E2 -16314.072} C_VEL
LIN {X 0,Y 311.031,Z 156.885,A -85,B 0,C 180,E1 -16315.015,E2 -16315.015} C_VEL
LIN {X 0,Y 306.736,Z 133.278,A -85,B 0,C 180,E1 -16315.987,E2 -16315.987} C_VEL
LIN {X 0,Y 302.252,Z 113.443,A -85,B 0,C 180,E1 -16316.951,E2 -16316.951} C_VEL
LIN {X 0,Y 302.147,Z 112.049,A -85,B 0,C 180,E1 -16317.348,E2 -16317.348} C_VEL
LIN {X 0,Y 300.96,Z 105.015,A -85,B 0,C 180,E1 -16320.228,E2 -16320.228} C_VEL
LIN {X 0,Y 299.397,Z 97.275,A -85,B 0,C 180,E1 -16323.479,E2 -16323.479} C_VEL
LIN {X 0,Y 298.475,Z 92.857,A -85,B 0,C 180,E1 -16325.45,E2 -16325.45} C_VEL
LIN {X 0,Y 298.411,Z 92.785,A -85,B 0,C 180,E1 -16329.486,E2 -16329.486} C_VEL
LIN {X 0,Y 298.401,Z 92.816,A -85,B 0,C 180,E1 -16333.103,E2 -16333.103} C_VEL
LIN {X 0,Y 298.405,Z 92.815,A -85,B 0,C 180,E1 -16336.92,E2 -16336.92} C_VEL
LIN {X 0,Y 298.406,Z 92.805,A -85,B 0,C 180,E1 -16341.006,E2 -16341.006} C_VEL
LIN {X 0,Y 298.42,Z 92.806,A -85,B 0,C 180,E1 -16343.93,E2 -16343.93} C_VEL
LIN {X 0,Y 298.395,Z 92.812,A -85,B 0,C 180,E1 -16347.983,E2 -16347.983} C_VEL
LIN {X 0,Y 298.46,Z 92.786,A -85,B 0,C 180,E1 -16351.903,E2 -16351.903} C_VEL
LIN {X 0,Y 298.487,Z 92.79,A -85,B 0,C 180,E1 -16354.923,E2 -16354.923} C_VEL
LIN {X 0,Y 298.451,Z 92.792,A -85,B 0,C 180,E1 -16359.315,E2 -16359.315} C_VEL
LIN {X 0,Y 298.538,Z 92.767,A -85,B 0,C 180,E1 -16362.179,E2 -16362.179} C_VEL
LIN {X 0,Y 298.594,Z 92.788,A -85,B 0,C 180,E1 -16364.994,E2 -16364.994} C_VEL
LIN {X 0,Y 298.594,Z 92.76,A -85,B 0,C 180,E1 -16369.146,E2 -16369.146} C_VEL
LIN {X 0,Y 298.76,Z 92.745,A -85,B 0,C 180,E1 -16371.885,E2 -16371.885} C_VEL
LIN {X 0,Y 298.661,Z 92.783,A -85,B 0,C 180,E1 -16374.598,E2 -16374.598} C_VEL
LIN {X 0,Y 298.922,Z 92.723,A -85,B 0,C 180,E1 -16378.652,E2 -16378.652} C_VEL
LIN {X 0,Y 298.922,Z 92.72,A -85,B 0,C 180,E1 -16381.346,E2 -16381.346} C_VEL
LIN {X 0,Y 298.797,Z 92.759,A -85,B 0,C 180,E1 -16386.753,E2 -16386.753} C_VEL
LIN {X 0,Y 298.68,Z 92.744,A -85,B 0,C 180,E1 -16389.48,E2 -16389.48} C_VEL
LIN {X 0,Y 298.553,Z 92.794,A -85,B 0,C 180,E1 -16393.615,E2 -16393.615} C_VEL
LIN {X 0,Y 298.547,Z 92.789,A -85,B 0,C 180,E1 -16396.408,E2 -16396.408} C_VEL
LIN {X 0,Y 298.51,Z 92.771,A -85,B 0,C 180,E1 -16399.654,E2 -16399.654} C_VEL
LIN {X 0,Y 298.456,Z 92.808,A -85,B 0,C 180,E1 -16403.597,E2 -16403.597} C_VEL
LIN {X 0,Y 298.484,Z 92.78,A -85,B 0,C 180,E1 -16406.574,E2 -16406.574} C_VEL
LIN {X 0,Y 298.414,Z 92.809,A -85,B 0,C 180,E1 -16409.641,E2 -16409.641} C_VEL
LIN {X 0,Y 298.392,Z 92.806,A -85,B 0,C 180,E1 -16412.8,E2 -16412.8} C_VEL
LIN {X 0,Y 298.463,Z 92.805,A -85,B 0,C 180,E1 -16416.812,E2 -16416.812} C_VEL
LIN {X 0,Y 298.414,Z 92.798,A -85,B 0,C 180,E1 -16421.094,E2 -16421.094} C_VEL
LIN {X 0,Y 298.423,Z 92.813,A -85,B 0,C 180,E1 -16423.108,E2 -16423.108} C_VEL
LIN {X 0,Y 298.399,Z 92.767,A -85,B 0,C 180,E1 -16426.92,E2 -16426.92} C_VEL
LIN {X 0,Y 298.411,Z 92.807,A -85,B 0,C 180,E1 -16431.003,E2 -16431.003} C_VEL
LIN {X 0,Y 298.428,Z 92.787,A -85,B 0,C 180,E1 -16433.932,E2 -16433.932} C_VEL
LIN {X 0,Y 298.391,Z 92.817,A -85,B 0,C 180,E1 -16437.983,E2 -16437.983} C_VEL
LIN {X 0,Y 298.487,Z 92.895,A -85,B 0,C 180,E1 -16442.273,E2 -16442.273} C_VEL
LIN {X 0,Y 298.652,Z 93.677,A -85,B 0,C 180,E1 -16442.54,E2 -16442.54} C_VEL
LIN {X 0,Y 300.885,Z 98.356,A -85,B 0,C 180,E1 -16442.936,E2 -16442.936} C_VEL
LIN {X 0,Y 306.849,Z 107.764,A -85,B 0,C 180,E1 -16443.777,E2 -16443.777} C_VEL
LIN {X 0,Y 311.971,Z 114.444,A -85,B 0,C 180,E1 -16444.513,E2 -16444.513} C_VEL
LIN {X 0,Y 317.601,Z 120.927,A -85,B 0,C 180,E1 -16445.379,E2 -16445.379} C_VEL
LIN {X 0,Y 322.752,Z 126.651,A -85,B 0,C 180,E1 -16446.244,E2 -16446.244} C_VEL
LIN {X 0,Y 328.372,Z 132.708,A -85,B 0,C 180,E1 -16447.287,E2 -16447.287} C_VEL
LIN {X 0,Y 335.007,Z 139.426,A -85,B 0,C 180,E1 -16448.625,E2 -16448.625} C_VEL
LIN {X 0,Y 341.491,Z 145.771,A -85,B 0,C 180,E1 -16450.031,E2 -16450.031} C_VEL
LIN {X 0,Y 349.033,Z 152.6,A -85,B 0,C 180,E1 -16451.818,E2 -16451.818} C_VEL
LIN {X 0,Y 353.426,Z 156.21,A -85,B 0,C 180,E1 -16452.936,E2 -16452.936} C_VEL
LIN {X 0,Y 358.491,Z 160.586,A -85,B 0,C 180,E1 -16454.351,E2 -16454.351} C_VEL
LIN {X 0,Y 362.862,Z 164.004,A -85,B 0,C 180,E1 -16455.68,E2 -16455.68} C_VEL
LIN {X 0,Y 367.469,Z 167.889,A -85,B 0,C 180,E1 -16457.261,E2 -16457.261} C_VEL
LIN {X 0,Y 371.535,Z 170.465,A -85,B 0,C 180,E1 -16458.81,E2 -16458.81} C_VEL
LIN {X 0,Y 373.558,Z 171.939,A -85,B 0,C 180,E1 -16459.672,E2 -16459.672} C_VEL
LIN {X 0,Y 377.053,Z 175.107,A -85,B 0,C 180,E1 -16461.424,E2 -16461.424} C_VEL
LIN {X 0,Y 380.083,Z 177.16,A -85,B 0,C 180,E1 -16463.274,E2 -16463.274} C_VEL
LIN {X 0,Y 382.595,Z 178.444,A -85,B 0,C 180,E1 -16465.263,E2 -16465.263} C_VEL
LIN {X 0,Y 384.297,Z 179.053,A -85,B 0,C 180,E1 -16467.367,E2 -16467.367} C_VEL
LIN {X 0,Y 384.936,Z 179.507,A -85,B 0,C 180,E1 -16468.954,E2 -16468.954} C_VEL
LIN {X 0,Y 385.081,Z 179.416,A -85,B 0,C 180,E1 -16470,E2 -16470} C_VEL
LIN {X 0,Y 384.785,Z 179.35,A -85,B 0,C 180,E1 -16471.57,E2 -16471.57} C_VEL
LIN {X 0,Y 383.978,Z 178.899,A -85,B 0,C 180,E1 -16473.148,E2 -16473.148} C_VEL
LIN {X 0,Y 382.282,Z 178.327,A -85,B 0,C 180,E1 -16475.001,E2 -16475.001} C_VEL
LIN {X 0,Y 379.791,Z 176.992,A -85,B 0,C 180,E1 -16476.927,E2 -16476.927} C_VEL
LIN {X 0,Y 376.552,Z 174.733,A -85,B 0,C 180,E1 -16478.839,E2 -16478.839} C_VEL
LIN {X 0,Y 372.815,Z 171.208,A -85,B 0,C 180,E1 -16480.664,E2 -16480.664} C_VEL
LIN {X 0,Y 368.428,Z 168.566,A -85,B 0,C 180,E1 -16482.386,E2 -16482.386} C_VEL
LIN {X 0,Y 364.109,Z 165.15,A -85,B 0,C 180,E1 -16483.901,E2 -16483.901} C_VEL
LIN {X 0,Y 359.981,Z 161.671,A -85,B 0,C 180,E1 -16485.208,E2 -16485.208} C_VEL
LIN {X 0,Y 354.625,Z 157.386,A -85,B 0,C 180,E1 -16486.732,E2 -16486.732} C_VEL
LIN {X 0,Y 350.408,Z 153.629,A -85,B 0,C 180,E1 -16487.849,E2 -16487.849} C_VEL
LIN {X 0,Y 345.168,Z 149.095,A -85,B 0,C 180,E1 -16489.127,E2 -16489.127} C_VEL
LIN {X 0,Y 338.01,Z 142.519,A -85,B 0,C 180,E1 -16490.729,E2 -16490.729} C_VEL
LIN {X 0,Y 330.471,Z 134.948,A -85,B 0,C 180,E1 -16492.294,E2 -16492.294} C_VEL
LIN {X 0,Y 323.735,Z 127.805,A -85,B 0,C 180,E1 -16493.572,E2 -16493.572} C_VEL
LIN {X 0,Y 317.929,Z 121.31,A -85,B 0,C 180,E1 -16494.569,E2 -16494.569} C_VEL
LIN {X 0,Y 312.876,Z 115.389,A -85,B 0,C 180,E1 -16495.357,E2 -16495.357} C_VEL
LIN {X 0,Y 308.932,Z 110.561,A -85,B 0,C 180,E1 -16495.934,E2 -16495.934} C_VEL
LIN {X 0,Y 302.671,Z 101.385,A -85,B 0,C 180,E1 -16496.811,E2 -16496.811} C_VEL
LIN {X 0,Y 298.712,Z 93.902,A -85,B 0,C 180,E1 -16497.429,E2 -16497.429} C_VEL
LIN {X 0,Y 298.487,Z 92.9,A -85,B 0,C 180,E1 -16497.727,E2 -16497.727} C_VEL
LIN {X 0,Y 298.391,Z 92.817,A -85,B 0,C 180,E1 -16502.017,E2 -16502.017} C_VEL
LIN {X 0,Y 298.428,Z 92.786,A -85,B 0,C 180,E1 -16506.068,E2 -16506.068} C_VEL
LIN {X 0,Y 298.405,Z 92.799,A -85,B 0,C 180,E1 -16509.487,E2 -16509.487} C_VEL
LIN {X 0,Y 298.395,Z 92.768,A -85,B 0,C 180,E1 -16513.104,E2 -16513.104} C_VEL
LIN {X 0,Y 298.4,Z 92.816,A -85,B 0,C 180,E1 -16516.921,E2 -16516.921} C_VEL
LIN {X 0,Y 298.423,Z 92.806,A -85,B 0,C 180,E1 -16521.002,E2 -16521.002} C_VEL
LIN {X 0,Y 298.43,Z 92.804,A -85,B 0,C 180,E1 -16523.933,E2 -16523.933} C_VEL
LIN {X 0,Y 298.391,Z 92.815,A -85,B 0,C 180,E1 -16527.984,E2 -16527.984} C_VEL
LIN {X 0,Y 298.456,Z 92.785,A -85,B 0,C 180,E1 -16531.904,E2 -16531.904} C_VEL
LIN {X 0,Y 298.483,Z 92.795,A -85,B 0,C 180,E1 -16534.925,E2 -16534.925} C_VEL
LIN {X 0,Y 298.448,Z 92.792,A -85,B 0,C 180,E1 -16539.316,E2 -16539.316} C_VEL
LIN {X 0,Y 298.536,Z 92.773,A -85,B 0,C 180,E1 -16542.18,E2 -16542.18} C_VEL
LIN {X 0,Y 298.593,Z 92.791,A -85,B 0,C 180,E1 -16544.996,E2 -16544.996} C_VEL
LIN {X 0,Y 298.594,Z 92.76,A -85,B 0,C 180,E1 -16549.147,E2 -16549.147} C_VEL
LIN {X 0,Y 298.758,Z 92.748,A -85,B 0,C 180,E1 -16551.887,E2 -16551.887} C_VEL
LIN {X 0,Y 298.659,Z 92.783,A -85,B 0,C 180,E1 -16554.6,E2 -16554.6} C_VEL
LIN {X 0,Y 298.922,Z 92.72,A -85,B 0,C 180,E1 -16558.654,E2 -16558.654} C_VEL
LIN {X 0,Y 298.922,Z 92.723,A -85,B 0,C 180,E1 -16561.348,E2 -16561.348} C_VEL
LIN {X 0,Y 298.8,Z 92.757,A -85,B 0,C 180,E1 -16566.755,E2 -16566.755} C_VEL
LIN {X 0,Y 298.755,Z 92.747,A -85,B 0,C 180,E1 -16567.895,E2 -16567.895} C_VEL
LIN {X 0,Y 298.073,Z 92.827,A -85,B 0,C 180,E1 -16569.019,E2 -16569.019} C_VEL
LIN {X 0,Y 295.112,Z 93.197,A -85,B 0,C 180,E1 -16570.844,E2 -16570.844} C_VEL
LIN {X 0,Y 292.618,Z 93.522,A -85,B 0,C 180,E1 -16572.327,E2 -16572.327} C_VEL
LIN {X 0,Y 291.582,Z 93.659,A -85,B 0,C 180,E1 -16573.478,E2 -16573.478} C_VEL
LIN {X 0,Y 291.518,Z 93.669,A -85,B 0,C 180,E1 -16573.868,E2 -16573.868} C_VEL
LIN {X 0,Y 291.488,Z 93.657,A -85,B 0,C 180,E1 -16576.819,E2 -16576.819} C_VEL
LIN {X 0,Y 291.452,Z 93.65,A -85,B 0,C 180,E1 -16579.876,E2 -16579.876} C_VEL
LIN {X 0,Y 291.402,Z 93.681,A -85,B 0,C 180,E1 -16584.206,E2 -16584.206} C_VEL
LIN {X 0,Y 291.421,Z 93.656,A -85,B 0,C 180,E1 -16587.272,E2 -16587.272} C_VEL
LIN {X 0,Y 291.336,Z 93.694,A -85,B 0,C 180,E1 -16590.438,E2 -16590.438} C_VEL
LIN {X 0,Y 291.346,Z 93.672,A -85,B 0,C 180,E1 -16593.699,E2 -16593.699} C_VEL
LIN {X 0,Y 291.378,Z 93.691,A -85,B 0,C 180,E1 -16597.255,E2 -16597.255} C_VEL
LIN {X 0,Y 291.334,Z 93.681,A -85,B 0,C 180,E1 -16600.643,E2 -16600.643} C_VEL
LIN {X 0,Y 291.292,Z 93.691,A -85,B 0,C 180,E1 -16604.402,E2 -16604.402} C_VEL
LIN {X 0,Y 291.328,Z 93.676,A -85,B 0,C 180,E1 -16608.405,E2 -16608.405} C_VEL
LIN {X 0,Y 291.367,Z 93.669,A -85,B 0,C 180,E1 -16611.161,E2 -16611.161} C_VEL
LIN {X 0,Y 291.428,Z 93.802,A -85,B 0,C 180,E1 -16614.104,E2 -16614.104} C_VEL
LIN {X 0,Y 293.113,Z 101.833,A -85,B 0,C 180,E1 -16617.667,E2 -16617.667} C_VEL
LIN {X 0,Y 294.837,Z 110.888,A -85,B 0,C 180,E1 -16621.528,E2 -16621.528} C_VEL
LIN {X 0,Y 295.218,Z 113.131,A -85,B 0,C 180,E1 -16622.338,E2 -16622.338} C_VEL
LIN {X 0,Y 296.971,Z 119.187,A -85,B 0,C 180,E1 -16622.725,E2 -16622.725} C_VEL
LIN {X 0,Y 302.105,Z 143.289,A -85,B 0,C 180,E1 -16623.847,E2 -16623.847} C_VEL
LIN {X 0,Y 304.672,Z 159.134,A -85,B 0,C 180,E1 -16624.488,E2 -16624.488} C_VEL
LIN {X 0,Y 303.102,Z 219.1,A -85,B 0,C 180,E1 -16625.924,E2 -16625.924} C_VEL
LIN {X 0,Y 302.453,Z 229.412,A -85,B 0,C 180,E1 -16626.324,E2 -16626.324} C_VEL
LIN {X 0,Y 301.544,Z 238.923,A -85,B 0,C 180,E1 -16626.84,E2 -16626.84} C_VEL
LIN {X 0,Y 300.482,Z 249.004,A -85,B 0,C 180,E1 -16627.571,E2 -16627.571} C_VEL
LIN {X 0,Y 299.194,Z 258.76,A -85,B 0,C 180,E1 -16628.468,E2 -16628.468} C_VEL
LIN {X 0,Y 297.678,Z 268.824,A -85,B 0,C 180,E1 -16629.62,E2 -16629.62} C_VEL
LIN {X 0,Y 295.804,Z 280.322,A -85,B 0,C 180,E1 -16631.292,E2 -16631.292} C_VEL
LIN {X 0,Y 294.332,Z 289.304,A -85,B 0,C 180,E1 -16632.958,E2 -16632.958} C_VEL
LIN {X 0,Y 293.207,Z 295.662,A -85,B 0,C 180,E1 -16634.356,E2 -16634.356} C_VEL
LIN {X 0,Y 292.072,Z 302.2,A -85,B 0,C 180,E1 -16636.077,E2 -16636.077} C_VEL
LIN {X 0,Y 291.242,Z 306.7,A -85,B 0,C 180,E1 -16637.457,E2 -16637.457} C_VEL
LIN {X 0,Y 290.424,Z 312.194,A -85,B 0,C 180,E1 -16639.543,E2 -16639.543} C_VEL
LIN {X 0,Y 289.857,Z 316.521,A -85,B 0,C 180,E1 -16641.635,E2 -16641.635} C_VEL
LIN {X 0,Y 289.609,Z 318.889,A -85,B 0,C 180,E1 -16643.031,E2 -16643.031} C_VEL
LIN {X 0,Y 289.436,Z 320.911,A -85,B 0,C 180,E1 -16644.599,E2 -16644.599} C_VEL
LIN {X 0,Y 289.431,Z 323.14,A -85,B 0,C 180,E1 -16647.216,E2 -16647.216} C_VEL
LIN {X 0,Y 289.408,Z 323.73,A -85,B 0,C 180,E1 -16648.608,E2 -16648.608} C_VEL
LIN {X 0,Y 289.408,Z 323.73,A -85,B 0,C 180,E1 -16651.392,E2 -16651.392} C_VEL
LIN {X 0,Y 289.431,Z 323.14,A -85,B 0,C 180,E1 -16652.784,E2 -16652.784} C_VEL
LIN {X 0,Y 289.479,Z 320.69,A -85,B 0,C 180,E1 -16655.573,E2 -16655.573} C_VEL
LIN {X 0,Y 289.721,Z 317.738,A -85,B 0,C 180,E1 -16657.667,E2 -16657.667} C_VEL
LIN {X 0,Y 290.192,Z 313.748,A -85,B 0,C 180,E1 -16659.76,E2 -16659.76} C_VEL
LIN {X 0,Y 290.932,Z 308.616,A -85,B 0,C 180,E1 -16661.849,E2 -16661.849} C_VEL
LIN {X 0,Y 291.871,Z 303.356,A -85,B 0,C 180,E1 -16663.578,E2 -16663.578} C_VEL
LIN {X 0,Y 292.97,Z 297.039,A -85,B 0,C 180,E1 -16665.3,E2 -16665.3} C_VEL
LIN {X 0,Y 294.301,Z 289.946,A -85,B 0,C 180,E1 -16666.904,E2 -16666.904} C_VEL
LIN {X 0,Y 295.502,Z 282.242,A -85,B 0,C 180,E1 -16668.368,E2 -16668.368} C_VEL
LIN {X 0,Y 296.918,Z 273.714,A -85,B 0,C 180,E1 -16669.712,E2 -16669.712} C_VEL
LIN {X 0,Y 298.59,Z 263.421,A -85,B 0,C 180,E1 -16671.035,E2 -16671.035} C_VEL
LIN {X 0,Y 300.204,Z 251.017,A -85,B 0,C 180,E1 -16672.269,E2 -16672.269} C_VEL
LIN {X 0,Y 301.448,Z 240.212,A -85,B 0,C 180,E1 -16673.077,E2 -16673.077} C_VEL
LIN {X 0,Y 302.385,Z 230.286,A -85,B 0,C 180,E1 -16673.636,E2 -16673.636} C_VEL
LIN {X 0,Y 302.968,Z 220.429,A -85,B 0,C 180,E1 -16674.042,E2 -16674.042} C_VEL
LIN {X 0,Y 303.687,Z 197.608,A -85,B 0,C 180,E1 -16674.618,E2 -16674.618} C_VEL
LIN {X 0,Y 304.584,Z 157.763,A -85,B 0,C 180,E1 -16675.555,E2 -16675.555} C_VEL
LIN {X 0,Y 300.227,Z 133.935,A -85,B 0,C 180,E1 -16676.572,E2 -16676.572} C_VEL
LIN {X 0,Y 296.083,Z 115.903,A -85,B 0,C 180,E1 -16677.451,E2 -16677.451} C_VEL
LIN {X 0,Y 295.19,Z 112.916,A -85,B 0,C 180,E1 -16677.701,E2 -16677.701} C_VEL
LIN {X 0,Y 293.681,Z 104.713,A -85,B 0,C 180,E1 -16681.095,E2 -16681.095} C_VEL
LIN {X 0,Y 292.185,Z 97.389,A -85,B 0,C 180,E1 -16684.287,E2 -16684.287} C_VEL
LIN {X 0,Y 291.418,Z 93.708,A -85,B 0,C 180,E1 -16686.004,E2 -16686.004} C_VEL
LIN {X 0,Y 291.389,Z 93.659,A -85,B 0,C 180,E1 -16689.483,E2 -16689.483} C_VEL
LIN {X 0,Y 291.311,Z 93.698,A -85,B 0,C 180,E1 -16693.633,E2 -16693.633} C_VEL
LIN {X 0,Y 291.322,Z 93.699,A -85,B 0,C 180,E1 -16697.507,E2 -16697.507} C_VEL
LIN {X 0,Y 291.355,Z 93.684,A -85,B 0,C 180,E1 -16701.158,E2 -16701.158} C_VEL
LIN {X 0,Y 291.363,Z 93.675,A -85,B 0,C 180,E1 -16704.625,E2 -16704.625} C_VEL
LIN {X 0,Y 291.372,Z 93.687,A -85,B 0,C 180,E1 -16707.95,E2 -16707.95} C_VEL
LIN {X 0,Y 291.379,Z 93.676,A -85,B 0,C 180,E1 -16711.157,E2 -16711.157} C_VEL
LIN {X 0,Y 291.416,Z 93.665,A -85,B 0,C 180,E1 -16714.271,E2 -16714.271} C_VEL
LIN {X 0,Y 291.383,Z 93.686,A -85,B 0,C 180,E1 -16717.299,E2 -16717.299} C_VEL
LIN {X 0,Y 291.459,Z 93.647,A -85,B 0,C 180,E1 -16720.269,E2 -16720.269} C_VEL
LIN {X 0,Y 291.556,Z 93.662,A -85,B 0,C 180,E1 -16724.623,E2 -16724.623} C_VEL
LIN {X 0,Y 291.537,Z 93.642,A -85,B 0,C 180,E1 -16728.88,E2 -16728.88} C_VEL
LIN {X 0,Y 291.71,Z 93.62,A -85,B 0,C 180,E1 -16731.688,E2 -16731.688} C_VEL
LIN {X 0,Y 291.632,Z 93.659,A -85,B 0,C 180,E1 -16734.468,E2 -16734.468} C_VEL
LIN {X 0,Y 291.888,Z 93.599,A -85,B 0,C 180,E1 -16738.62,E2 -16738.62} C_VEL
LIN {X 0,Y 291.888,Z 93.596,A -85,B 0,C 180,E1 -16741.379,E2 -16741.379} C_VEL
LIN {X 0,Y 291.746,Z 93.636,A -85,B 0,C 180,E1 -16746.917,E2 -16746.917} C_VEL
LIN {X 0,Y 291.629,Z 93.621,A -85,B 0,C 180,E1 -16749.711,E2 -16749.711} C_VEL
LIN {X 0,Y 291.522,Z 93.672,A -85,B 0,C 180,E1 -16753.949,E2 -16753.949} C_VEL
LIN {X 0,Y 291.486,Z 93.662,A -85,B 0,C 180,E1 -16756.817,E2 -16756.817} C_VEL
LIN {X 0,Y 291.449,Z 93.651,A -85,B 0,C 180,E1 -16759.874,E2 -16759.874} C_VEL
LIN {X 0,Y 291.399,Z 93.685,A -85,B 0,C 180,E1 -16764.205,E2 -16764.205} C_VEL
LIN {X 0,Y 291.418,Z 93.657,A -85,B 0,C 180,E1 -16767.271,E2 -16767.271} C_VEL
LIN {X 0,Y 291.332,Z 93.694,A -85,B 0,C 180,E1 -16770.437,E2 -16770.437} C_VEL
LIN {X 0,Y 291.342,Z 93.676,A -85,B 0,C 180,E1 -16773.698,E2 -16773.698} C_VEL
LIN {X 0,Y 291.396,Z 93.689,A -85,B 0,C 180,E1 -16777.259,E2 -16777.259} C_VEL
LIN {X 0,Y 291.373,Z 93.674,A -85,B 0,C 180,E1 -16780.635,E2 -16780.635} C_VEL
LIN {X 0,Y 291.295,Z 93.694,A -85,B 0,C 180,E1 -16784.4,E2 -16784.4} C_VEL
LIN {X 0,Y 291.322,Z 93.643,A -85,B 0,C 180,E1 -16788.404,E2 -16788.404} C_VEL
LIN {X 0,Y 291.361,Z 93.687,A -85,B 0,C 180,E1 -16791.16,E2 -16791.16} C_VEL
LIN {X 0,Y 291.381,Z 93.656,A -85,B 0,C 180,E1 -16794.629,E2 -16794.629} C_VEL
LIN {X 0,Y 291.368,Z 93.691,A -85,B 0,C 180,E1 -16797.95,E2 -16797.95} C_VEL
LIN {X 0,Y 291.423,Z 93.827,A -85,B 0,C 180,E1 -16801.615,E2 -16801.615} C_VEL
LIN {X 0,Y 291.691,Z 94.934,A -85,B 0,C 180,E1 -16801.893,E2 -16801.893} C_VEL
LIN {X 0,Y 298.162,Z 106.949,A -85,B 0,C 180,E1 -16802.895,E2 -16802.895} C_VEL
LIN {X 0,Y 305.941,Z 117.798,A -85,B 0,C 180,E1 -16803.946,E2 -16803.946} C_VEL
LIN {X 0,Y 312.905,Z 125.747,A -85,B 0,C 180,E1 -16804.929,E2 -16804.929} C_VEL
LIN {X 0,Y 318.858,Z 132.2,A -85,B 0,C 180,E1 -16805.858,E2 -16805.858} C_VEL
LIN {X 0,Y 324.613,Z 138.287,A -85,B 0,C 180,E1 -16806.867,E2 -16806.867} C_VEL
LIN {X 0,Y 331.289,Z 144.913,A -85,B 0,C 180,E1 -16808.141,E2 -16808.141} C_VEL
LIN {X 0,Y 338.973,Z 152.202,A -85,B 0,C 180,E1 -16809.745,E2 -16809.745} C_VEL
LIN {X 0,Y 346.401,Z 158.824,A -85,B 0,C 180,E1 -16811.455,E2 -16811.455} C_VEL
LIN {X 0,Y 350.974,Z 162.532,A -85,B 0,C 180,E1 -16812.589,E2 -16812.589} C_VEL
LIN {X 0,Y 356.404,Z 167.137,A -85,B 0,C 180,E1 -16814.063,E2 -16814.063} C_VEL
LIN {X 0,Y 360.801,Z 170.485,A -85,B 0,C 180,E1 -16815.365,E2 -16815.365} C_VEL
LIN {X 0,Y 365.507,Z 174.38,A -85,B 0,C 180,E1 -16816.91,E2 -16816.91} C_VEL
LIN {X 0,Y 369.816,Z 177.148,A -85,B 0,C 180,E1 -16818.498,E2 -16818.498} C_VEL
LIN {X 0,Y 372.051,Z 178.69,A -85,B 0,C 180,E1 -16819.425,E2 -16819.425} C_VEL
LIN {X 0,Y 375.289,Z 181.585,A -85,B 0,C 180,E1 -16820.977,E2 -16820.977} C_VEL
LIN {X 0,Y 378.558,Z 183.872,A -85,B 0,C 180,E1 -16822.854,E2 -16822.854} C_VEL
LIN {X 0,Y 381.112,Z 185.202,A -85,B 0,C 180,E1 -16824.74,E2 -16824.74} C_VEL
LIN {X 0,Y 382.566,Z 185.759,A -85,B 0,C 180,E1 -16826.158,E2 -16826.158} C_VEL
LIN {X 0,Y 383.703,Z 186.233,A -85,B 0,C 180,E1 -16827.901,E2 -16827.901} C_VEL
LIN {X 0,Y 384.071,Z 186.553,A -85,B 0,C 180,E1 -16828.952,E2 -16828.952} C_VEL
LIN {X 0,Y 384.216,Z 186.463,A -85,B 0,C 180,E1 -16830,E2 -16830} C_VEL
LIN {X 0,Y 383.919,Z 186.382,A -85,B 0,C 180,E1 -16831.573,E2 -16831.573} C_VEL
LIN {X 0,Y 383.103,Z 185.923,A -85,B 0,C 180,E1 -16833.155,E2 -16833.155} C_VEL
LIN {X 0,Y 381.392,Z 185.373,A -85,B 0,C 180,E1 -16835.012,E2 -16835.012} C_VEL
LIN {X 0,Y 378.868,Z 184.054,A -85,B 0,C 180,E1 -16836.944,E2 -16836.944} C_VEL
LIN {X 0,Y 375.719,Z 181.933,A -85,B 0,C 180,E1 -16838.793,E2 -16838.793} C_VEL
LIN {X 0,Y 372.535,Z 179.155,A -85,B 0,C 180,E1 -16840.357,E2 -16840.357} C_VEL
LIN {X 0,Y 370.158,Z 177.333,A -85,B 0,C 180,E1 -16841.365,E2 -16841.365} C_VEL
LIN {X 0,Y 365.702,Z 174.507,A -85,B 0,C 180,E1 -16843.021,E2 -16843.021} C_VEL
LIN {X 0,Y 360.855,Z 170.554,A -85,B 0,C 180,E1 -16844.618,E2 -16844.618} C_VEL
LIN {X 0,Y 356.852,Z 167.441,A -85,B 0,C 180,E1 -16845.814,E2 -16845.814} C_VEL
LIN {X 0,Y 351.4,Z 162.937,A -85,B 0,C 180,E1 -16847.299,E2 -16847.299} C_VEL
LIN {X 0,Y 347.91,Z 159.963,A -85,B 0,C 180,E1 -16848.182,E2 -16848.182} C_VEL
LIN {X 0,Y 342.748,Z 155.583,A -85,B 0,C 180,E1 -16849.402,E2 -16849.402} C_VEL
LIN {X 0,Y 335.125,Z 148.705,A -85,B 0,C 180,E1 -16851.068,E2 -16851.068} C_VEL
LIN {X 0,Y 327.039,Z 140.745,A -85,B 0,C 180,E1 -16852.684,E2 -16852.684} C_VEL
LIN {X 0,Y 320.372,Z 133.92,A -85,B 0,C 180,E1 -16853.88,E2 -16853.88} C_VEL
LIN {X 0,Y 312.533,Z 125.409,A -85,B 0,C 180,E1 -16855.126,E2 -16855.126} C_VEL
LIN {X 0,Y 304.74,Z 116.285,A -85,B 0,C 180,E1 -16856.218,E2 -16856.218} C_VEL
LIN {X 0,Y 297.45,Z 105.723,A -85,B 0,C 180,E1 -16857.209,E2 -16857.209} C_VEL
LIN {X 0,Y 291.645,Z 94.777,A -85,B 0,C 180,E1 -16858.13,E2 -16858.13} C_VEL
LIN {X 0,Y 291.407,Z 93.751,A -85,B 0,C 180,E1 -16858.451,E2 -16858.451} C_VEL
LIN {X 0,Y 291.34,Z 93.686,A -85,B 0,C 180,E1 -16862.404,E2 -16862.404} C_VEL
LIN {X 0,Y 291.381,Z 93.655,A -85,B 0,C 180,E1 -16865.371,E2 -16865.371} C_VEL
LIN {X 0,Y 291.361,Z 93.687,A -85,B 0,C 180,E1 -16868.84,E2 -16868.84} C_VEL
LIN {X 0,Y 291.315,Z 93.643,A -85,B 0,C 180,E1 -16872.493,E2 -16872.493} C_VEL
LIN {X 0,Y 291.326,Z 93.696,A -85,B 0,C 180,E1 -16876.363,E2 -16876.363} C_VEL
LIN {X 0,Y 291.392,Z 93.679,A -85,B 0,C 180,E1 -16880.515,E2 -16880.515} C_VEL
LIN {X 0,Y 291.425,Z 93.685,A -85,B 0,C 180,E1 -16882.923,E2 -16882.923} C_VEL
LIN {X 0,Y 291.342,Z 93.676,A -85,B 0,C 180,E1 -16886.302,E2 -16886.302} C_VEL
LIN {X 0,Y 291.381,Z 93.686,A -85,B 0,C 180,E1 -16890.262,E2 -16890.262} C_VEL
LIN {X 0,Y 291.412,Z 93.67,A -85,B 0,C 180,E1 -16894.272,E2 -16894.272} C_VEL
LIN {X 0,Y 291.38,Z 93.687,A -85,B 0,C 180,E1 -16897.3,E2 -16897.3} C_VEL
LIN {X 0,Y 291.456,Z 93.649,A -85,B 0,C 180,E1 -16900.271,E2 -16900.271} C_VEL
LIN {X 0,Y 291.554,Z 93.666,A -85,B 0,C 180,E1 -16904.624,E2 -16904.624} C_VEL
LIN {X 0,Y 291.538,Z 93.641,A -85,B 0,C 180,E1 -16908.881,E2 -16908.881} C_VEL
LIN {X 0,Y 291.708,Z 93.623,A -85,B 0,C 180,E1 -16911.689,E2 -16911.689} C_VEL
LIN {X 0,Y 291.63,Z 93.66,A -85,B 0,C 180,E1 -16914.469,E2 -16914.469} C_VEL
LIN {X 0,Y 291.888,Z 93.596,A -85,B 0,C 180,E1 -16918.621,E2 -16918.621} C_VEL
LIN {X 0,Y 291.888,Z 93.599,A -85,B 0,C 180,E1 -16921.38,E2 -16921.38} C_VEL
LIN {X 0,Y 291.748,Z 93.634,A -85,B 0,C 180,E1 -16926.919,E2 -16926.919} C_VEL
LIN {X 0,Y 291.63,Z 93.619,A -85,B 0,C 180,E1 -16929.713,E2 -16929.713} C_VEL
LIN {X 0,Y 291.518,Z 93.669,A -85,B 0,C 180,E1 -16933.868,E2 -16933.868} C_VEL
LIN {X 0,Y 290.883,Z 93.753,A -85,B 0,C 180,E1 -16935.02,E2 -16935.02} C_VEL
LIN {X 0,Y 287.975,Z 94.097,A -85,B 0,C 180,E1 -16936.895,E2 -16936.895} C_VEL
LIN {X 0,Y 285.495,Z 94.389,A -85,B 0,C 180,E1 -16938.417,E2 -16938.417} C_VEL
LIN {X 0,Y 284.454,Z 94.518,A -85,B 0,C 180,E1 -16939.599,E2 -16939.599} C_VEL
LIN {X 0,Y 284.384,Z 94.531,A -85,B 0,C 180,E1 -16939.999,E2 -16939.999} C_VEL
LIN {X 0,Y 284.371,Z 94.558,A -85,B 0,C 180,E1 -16943.876,E2 -16943.876} C_VEL
LIN {X 0,Y 284.396,Z 94.53,A -85,B 0,C 180,E1 -16947.173,E2 -16947.173} C_VEL
LIN {X 0,Y 284.295,Z 94.571,A -85,B 0,C 180,E1 -16951.275,E2 -16951.275} C_VEL
LIN {X 0,Y 284.343,Z 94.549,A -85,B 0,C 180,E1 -16955.349,E2 -16955.349} C_VEL
LIN {X 0,Y 284.314,Z 94.57,A -85,B 0,C 180,E1 -16958.17,E2 -16958.17} C_VEL
LIN {X 0,Y 284.271,Z 94.574,A -85,B 0,C 180,E1 -16962.125,E2 -16962.125} C_VEL
LIN {X 0,Y 284.258,Z 94.575,A -85,B 0,C 180,E1 -16966.19,E2 -16966.19} C_VEL
LIN {X 0,Y 284.309,Z 94.538,A -85,B 0,C 180,E1 -16970.024,E2 -16970.024} C_VEL
LIN {X 0,Y 284.397,Z 94.627,A -85,B 0,C 180,E1 -16973.514,E2 -16973.514} C_VEL
LIN {X 0,Y 286.08,Z 102.837,A -85,B 0,C 180,E1 -16977.285,E2 -16977.285} C_VEL
LIN {X 0,Y 287.851,Z 112.101,A -85,B 0,C 180,E1 -16981.348,E2 -16981.348} C_VEL
LIN {X 0,Y 288.107,Z 113.284,A -85,B 0,C 180,E1 -16981.631,E2 -16981.631} C_VEL
LIN {X 0,Y 290.625,Z 120.431,A -85,B 0,C 180,E1 -16982.117,E2 -16982.117} C_VEL
LIN {X 0,Y 295.826,Z 144.933,A -85,B 0,C 180,E1 -16983.297,E2 -16983.297} C_VEL
LIN {X 0,Y 298.252,Z 159.635,A -85,B 0,C 180,E1 -16983.916,E2 -16983.916} C_VEL
LIN {X 0,Y 296.646,Z 218.914,A -85,B 0,C 180,E1 -16985.366,E2 -16985.366} C_VEL
LIN {X 0,Y 295.968,Z 229.222,A -85,B 0,C 180,E1 -16985.773,E2 -16985.773} C_VEL
LIN {X 0,Y 295.014,Z 238.732,A -85,B 0,C 180,E1 -16986.296,E2 -16986.296} C_VEL
LIN {X 0,Y 293.937,Z 248.814,A -85,B 0,C 180,E1 -16987.044,E2 -16987.044} C_VEL
LIN {X 0,Y 292.602,Z 258.569,A -85,B 0,C 180,E1 -16987.957,E2 -16987.957} C_VEL
LIN {X 0,Y 291.023,Z 268.633,A -85,B 0,C 180,E1 -16989.133,E2 -16989.133} C_VEL
LIN {X 0,Y 289.072,Z 280.131,A -85,B 0,C 180,E1 -16990.84,E2 -16990.84} C_VEL
LIN {X 0,Y 287.621,Z 288.274,A -85,B 0,C 180,E1 -16992.359,E2 -16992.359} C_VEL
LIN {X 0,Y 286.341,Z 295.471,A -85,B 0,C 180,E1 -16993.971,E2 -16993.971} C_VEL
LIN {X 0,Y 285.158,Z 302.009,A -85,B 0,C 180,E1 -16995.732,E2 -16995.732} C_VEL
LIN {X 0,Y 284.283,Z 306.509,A -85,B 0,C 180,E1 -16997.144,E2 -16997.144} C_VEL
LIN {X 0,Y 283.406,Z 312.002,A -85,B 0,C 180,E1 -16999.281,E2 -16999.281} C_VEL
LIN {X 0,Y 282.805,Z 316.329,A -85,B 0,C 180,E1 -17001.425,E2 -17001.425} C_VEL
LIN {X 0,Y 282.557,Z 318.698,A -85,B 0,C 180,E1 -17002.856,E2 -17002.856} C_VEL
LIN {X 0,Y 282.358,Z 320.939,A -85,B 0,C 180,E1 -17004.64,E2 -17004.64} C_VEL
LIN {X 0,Y 282.337,Z 322.95,A -85,B 0,C 180,E1 -17007.146,E2 -17007.146} C_VEL
